// TwinCAT 3 PLC project tc_project_app
// ProgramVersion: 3.1.4026.24
// libraries:
//   Tc2_EtherCAT, * (Beckhoff Automation GmbH)
//   Tc2_MC2, * (Beckhoff Automation GmbH)
//   Tc2_Standard, * (Beckhoff Automation GmbH)
//   Tc2_SUPS, * (Beckhoff Automation GmbH)
//   Tc2_System, * (Beckhoff Automation GmbH)
//   Tc2_Utilities, * (Beckhoff Automation GmbH)
//   Tc3_EventLogger, * (Beckhoff Automation GmbH)
//   Tc3_MC2_AdvancedHoming, * (Beckhoff Automation GmbH)
//   Tc3_Module, * (Beckhoff Automation GmbH)
//   VisuDialogs, * (System)
// project tree:
//   DUTs/ E_AxisNames.TcDUT, E_PendantControl.TcDUT, E_SWLimitControl.TcDUT, ST_PendantControl.TcDUT
//   / GlobalTextList.TcGTLO, PlcTask.TcTTO, Visualization Manager.TcVMO (not stored)
//   GVLs/ GVL_APP.TcGVL, KeTop.TcGVL
//   POUs/Application_Specific/Applications/ Application_Template.TcPOU (not stored), Pendant.TcPOU
//   POUs/Application_Specific/Axes/ Axis1.TcPOU, Axis_Template.TcPOU, Pneumatics_Template.TcPOU (not stored)
//   POUs/Application_Specific/Groups/ GROUP_1.TcPOU, Group_Template.TcPOU
//   POUs/ MAIN.TcPOU, PANEL.TcPOU, SAFETY.TcPOU
//   tc_mca_std_lib/DUTs/Axis_Group_Structures/ ST_AxisGroupDescription.TcDUT, ST_AxisGroupFlag.TcDUT, ST_AxisGroupStruct.TcDUT
//   tc_mca_std_lib/DUTs/Axis_Structures/ ST_AxisConfig.TcDUT, ST_AxisControl.TcDUT, ST_AxisDescription.TcDUT, ST_AxisError.TcDUT, ST_AxisHomingConfig.TcDUT, ST_AxisInputs.TcDUT, ST_AxisPersistent.TcDUT, ST_AxisSPG.TcDUT, ST_AxisStatus.TcDUT, ST_AxisStruct.TcDUT
//   tc_mca_std_lib/DUTs/ E_AxisParameters.TcTLEO, E_AxisParameters.TcTLEO, E_HomingRoutines.TcDUT, E_RestorePosition.TcDUT, E_SafetyType.TcDUT, I_Axis.TcIO, E_SlitPairStatesV2.TcDUT, E_SlitPairStates.TcDUT, E_MotionFunctions.TcDUT, ST_McStatus.TcDUT
//   tc_mca_std_lib/DUTs/Panel_Infrastructure/ ST_ECB.TcDUT
//   tc_mca_std_lib/DUTs/Pneumatics/ E_PneumaticAxisErrors.TcDUT, E_PneumaticMode.TcDUT, ST_PneumaticAxisControl.TcDUT, ST_PneumaticAxisConfig.TcDUT, ST_PneumaticAxisInputs.TcDUT, ST_PneumaticAxisOutputs.TcDUT, ST_PneumaticAxisStatus.TcDUT, ST_PneumaticAxisStruct.TcDUT
//   tc_mca_std_lib/DUTs/Safety_Structures/ ST_DeviceDualChannelInput.TcDUT, ST_DeviceSingleChannelInput.TcDUT, ST_SafetyDescription.TcDUT, ST_SafetyGroup.TcDUT, ST_SafetyTargetDevice.TcDUT
//   tc_mca_std_lib/GVLs/ GVL.TcGVL, GVL_UnitStrings.TcGVL
//   tc_mca_std_lib/POUs/Motion/ FB_Axis.TcPOU, FB_AxisGroups.TcPOU, FB_SlitPair.TcPOU, FB_SlitPairV2.TcPOU, FB_SlitPairV3.TcPOU
//   tc_mca_std_lib/POUs/Motion/Homing/ FB_Homing.TcPOU
//   tc_mca_std_lib/POUs/Pneumatics/ FB_PneumaticAxis.TcPOU
//   tc_mca_std_lib/VISUs/ MainVisu.TcVIS, ParameterTextList.TcTLO, PneumaticsVisu.TcVIS
// real-time tasks:
//   TASK PlcTask: cycle T#10ms, priority 10, ADS port 351
// motion (NC):
//   TASK NC-Task 1 SAF: cycle T#2ms, priority 4, ADS port 501
//   TASK NC-Task 1 SVB: cycle T#10ms, priority 8, ADS port 511
//   AXIS Axis1 (id 1)
//     Dynamic: AccelerationMaximum=60, DecelerationMaximum=60, Acceleration=12, Deceleration=12, Jerk=42
//     Velo: RefSearch=5, RefSync=0.2, SlowManual=1, FastManual=5, Fast=9.091, Maximum=6.5
//     TargetPosControl: Range=0.25, Time=0.2
//     OtherSettings: AllowMotionCmdToSlave=true
//     encoder EncType=1
//       EncPara: ScaleFactorNumerator=20, ScaleFactorDenominator=12582912, Inverse=true
//         SoftEndMinControl: Range=-300
//         SoftEndMaxControl: Range=300
//     drive DrvType=5
//       DrvPara: Inverse=true
//         Analog: VeloReferenz=10.0001, TorqueSetpointScale=10, ScaleFactorActTorque=0.1
//         TimeComp: TaskDelayCycles=1
//     controller CtrType=1
//       CtrPara: PriorControlFactor=1
//         PosDiffControl: Range=2
//         Observer: BandWidth=20
// variable links:
//   tc_project_app Instance <-> NC-Task 1 SAF/Axes/Axis1
//     PlcTask Inputs/GVL.astAxes[1].Axis.NcToPlc <-> Outputs/ToPlc
//     PlcTask Outputs/GVL.astAxes[1].Axis.PlcToNc <-> Inputs/FromPlc

CONFIGURATION tc_project_app
    RESOURCE PLC ON TwinCAT3
        TASK PlcTask(INTERVAL := T#10ms, PRIORITY := 10);
        PROGRAM MAIN WITH PlcTask : MAIN;
        PROGRAM SAFETY WITH PlcTask : SAFETY;
        PROGRAM PANEL WITH PlcTask : PANEL;
    END_RESOURCE
END_CONFIGURATION

// ---- DUTs/E_AxisNames.TcDUT
{attribute 'qualified_only'}
{attribute 'to_string'}
TYPE E_AxisNames :
(
	None := 0,
	IncSlits_X_Translation := 1,
	IncSlits_Z_Translation :=2,
	IncSlits_North := 3,
	IncSlits_South := 4,
	IncSlits_East := 5,
	IncSlits_West := 6,
	Sample_Stack_X_Translation := 7,
	Sample_Stack_Y_Translation := 8,
	Tomography_Phi := 9,
	Tomography_Chi := 10,
	Tomography_Theta := 11,
	SampleEnv_ExtraAxes := 12,
	Camera_LensAdj := 13,
	Camera_FlipRot := 14, // check correct
	Camera_Tilt := 15, //check correct
	Sample_Stack_Z_Translation :=16,
	Sample_Stack_Z_Rotation :=17,
	Coll_North_X :=18,
	Coll_North_Y :=19,
	Coll_South_X :=20,
	Coll_South_Y :=21,
	PinholeSelector := 22,
	Monitor5 := 23,
	Slit_1_North := 24,
	Slit_1_South := 25,
	Slit_1_East := 26,
	Slit_1_West := 27,
	Slit_2_North := 28,
	Slit_2_South := 29,
	Slit_2_East := 30,
	Slit_2_West := 31,
	Slit_3_North := 32,
	Slit_3_South := 33,
	Slit_3_East := 34,
	Slit_3_West := 35,
	Slit_4_North := 36,
	Slit_4_South := 37,
	Slit_4_East := 38,
	Slit_4_West := 39,
	Slit_5_North := 40,
	Slit_5_South := 41,
	Slit_5_East := 42,
	Slit_5_West := 43
);
END_TYPE

// ---- DUTs/E_PendantControl.TcDUT
{attribute 'qualified_only'}
TYPE E_PendantControl :
(
	Default := 0,
	JogFwd := 33,
	JogBwd := 32,
	SmallTweakFwd := 19,
	SmallTweakBwd := 25,
	MediumTweakFwd := 45,
	MediumTweakBwd := 47,
	BigTweakFwd := 5,
	BigTweakBwd := 3,	
	AbsMove := 15,
	Stop := 12,
    SlowJogFwd := 38,
    SlowJogBwd := 36,
	WaitForAbsoluteFinish := 127,
	WaitForJogFinish := 128,
    WaitForTweakFinish := 129,
	Error := 150
);
END_TYPE

// ---- DUTs/E_SWLimitControl.TcDUT
{attribute 'qualified_only'}
TYPE E_SWLimitControl :
(
	Default := 0,
	WriteFwdLimit := 1,
	WriteBwdLimit := 2,
	EnableSWLimits := 3,
	DisableSWLimits := 4
);
END_TYPE

// ---- DUTs/ST_PendantControl.TcDUT
TYPE ST_PendantControl :
STRUCT
	fTargetPosition : LREAL;
	fVelocity : LREAL := 100;
	fFwdLimit : LREAL;
	fBwdLimit : LREAL;
	fLocalModeSpeedOverride : LREAL;
END_STRUCT
END_TYPE

// ---- tc_mca_std_lib/DUTs/Axis_Group_Structures/ST_AxisGroupDescription.TcDUT
TYPE ST_AxisGroupDescription :
STRUCT
	sGroupName : STRING(nMAX_AXIS_GROUP_NAME);
	iAxesInGroup : INT;
END_STRUCT
END_TYPE

// ---- tc_mca_std_lib/DUTs/Axis_Group_Structures/ST_AxisGroupFlag.TcDUT
TYPE ST_AxisGroupFlag :
STRUCT
	iError : INT;
	iDisabled : INT;
	iState : INT;
	bErrorFlag : BOOL;
	bDisabledFlag : BOOL;
	iNumberOfAxisInError : INT;
	iNumberOfAxisDisabled : INT;
END_STRUCT
END_TYPE

// ---- tc_mca_std_lib/DUTs/Axis_Group_Structures/ST_AxisGroupStruct.TcDUT
TYPE ST_AxisGroupStruct :
STRUCT
	aAxesInGroup : ARRAY[1..GVL.nMAX_AXES_PER_GROUP] OF INT :=[GVL.nMAX_AXES_PER_GROUP(0)];
	stDescription : ST_AxisGroupDescription;
	stFlag : ST_AxisGroupFlag;
END_STRUCT
END_TYPE

// ---- tc_mca_std_lib/DUTs/Axis_Structures/ST_AxisConfig.TcDUT
(*These are axis parameters that are set up during commissioning and
in theory don't neeed to be change as part of daily moving of axes.
For instance they may be changed due to poor parameter selection
or change of instrument configuration.*)
TYPE ST_AxisConfig :
STRUCT
    //Axis Parameters
    fOverride: LREAL := 100; //Controller override %, used a global scale for an axis in terms of velocity. Generally set to 100%.
    
    eRestorePosition: E_RestorePosition; //Restore position of incremental axis after loss of power to the CPU, 0=don't restore, 1=restore but don't home

    //Read and Write parameters
    eAxisParameters: E_AxisParameters; //Enumeration of axis parameters
	fWriteAxisBoolParameter: BOOL; //The Bool value to be writen to eAxisParameterNumber
    fWriteAxisParameter: LREAL; //The value to be writen to eAxisParameterNumber
    fReadAxisParameter: LREAL; //Read the current value of the selected eAxisParameterNumber

    

    // Read only MC parameters
    bReadMcParametersValid: BOOL:= FALSE;
    bReadMcParametersError: BOOL:= FALSE;
    fVelocityDefaultSlow: LREAL; //Read only - AxisVeloManSlow
    fVelocityDefaultFast: LREAL; //Read only - AxisVeloManFast
    
    fVeloMax: LREAL; //Read only - AxisMaxVelocity
    fMaxAcc: LREAL; //Read only - AxisMaximumAcceleration
    fMaxDec: LREAL; //Read only - AxisMaxDeceleration
    fDefaultAcc: LREAL; //Read only - AxisDefaultAcceleration
    fDefaultDec: LREAL; //Read only - AxisDefaultDeceleration
    bEnMinSoftPosLimit: BOOL; //Read only
    fMinSoftPosLimit: LREAL; //Read only
    bEnMaxSoftPosLimit: BOOL; //Read only
    fMaxSoftPosLimit: LREAL; //Read only
    bEnPositionLagMonitoring: BOOL; //Read only
    fMaxPosLagValue: LREAL; //Read only
    bEnTargetPositionMonitoring: BOOL; //Read only
    fTargetPositionWindow: LREAL; //Read only
END_STRUCT
END_TYPE

// ---- tc_mca_std_lib/DUTs/Axis_Structures/ST_AxisControl.TcDUT
(*These are parameters that are used to initiate axis movements
They are commands that are commonly used commands*)
TYPE ST_AxisControl :
STRUCT
    //Actions from controls system
    bExecute: BOOL; //Rising edge to execute some motion FB's
    bReset: BOOL; //Reset axis from Error state
    bStop: BOOL;
    bHalt: BOOL;
    bEnable: BOOL; //Enable axis drive
    bJogFwd: BOOL;
    bJogBwd: BOOL;
    bInterlockFwd: BOOL := FALSE; //Bit for interlocking motors in the positive direction
    bInterlockBwd: BOOL := FALSE; //Bit for interlocking motors in the negative direction
    eCommand: E_MotionFunctions;
    fVelocity: LREAL; //Velocity must be specified
    fJogVelocity: LREAL; //Jogging velocity
    fAcceleration: LREAL; //Not all FBs use, 0 is NC default
    fDeceleration: LREAL;
    fPosition: LREAL; //The position to move to for an absolute move and the amount to move in a relative move
	fRelativePosition: LREAL; //Position for relative moves
	fSetPosition : LREAL;
	bReinitialiseNcParameters : BOOL;
	bWaitBeforeEnable : BOOL:= FALSE; //Code to allow 'other things' to happen before enabling axis when working with autoenabledisable logic
	bReadyToEnable : BOOL; //trigger signal for the above
	
	bOverrideLimits : BOOL;
	
	bAutoEnableDisable : BOOL;
	
	bOverrideReadyToMove : BOOL;
	bExtReadyToMove : BOOL;
	tMoveFinishedDelay : TIME := T#1S;
END_STRUCT
END_TYPE

// ---- tc_mca_std_lib/DUTs/Axis_Structures/ST_AxisDescription.TcDUT
TYPE ST_AxisDescription :
STRUCT
	iGroupNumber : INT;
    sUnits : STRING := UNIT_mm;
END_STRUCT
END_TYPE

// ---- tc_mca_std_lib/DUTs/Axis_Structures/ST_AxisError.TcDUT

TYPE ST_AxisError:
STRUCT
//PLCopen function block errors
    nPowerErrorID: UDINT;
    nMoveAbsoluteErrorID: UDINT;
	nLocalMoveAbsoluteErrorID: UDINT;
    nMoveRelativeErrorID: UDINT;
	nLocalMoveRelativeErrorID: UDINT;
    nMoveVelocityErrorID: UDINT;
	nLocalMoveVelocityErrorID: UDINT;
    nMoveModuloErrorID: UDINT;
    nJogErrorID: UDINT;
    nHomeErrorID: UDINT;
    nHaltErrorID: UDINT;
    nResetErrorID: UDINT;
    nStopErrorID: UDINT;
    nGearInMultiMasterErrorID: UDINT;
    nGearOutErrorID: UDINT;
	nSetPositionErrorID : UDINT;
    fbWriteParameterErrorId: UDINT;
    fbReadParameterErrorId: UDINT;
//Error from the NC
    nNCErrorID : UDINT;
END_STRUCT
END_TYPE

// ---- tc_mca_std_lib/DUTs/Axis_Structures/ST_AxisHomingConfig.TcDUT
TYPE ST_AxisHomingConfig :
STRUCT
	fHomePosition: LREAL := 0; //The position that the axis should be set to once homing is completed
    fHomeFinishDistance: LREAL := 0; //Distrance that the axis should move back into the working zone after homing is finished
    eHomeSeq: E_HomingRoutines; //Homing sequence to perform
	fHomeAbsPosition : LREAL:= 0;
	fHomeMidRelativeMove : LREAL:= 1;
	
	bGoToFwdFirst : BOOL; //Takes priority over bwd bool, optional command to go to fwd limit before homing
	bGoToBwdFirst : BOOL; //optional command to go to bwd limit before homing
	bDoAbsoluteMoveAtEnd : BOOL;
	
	
	//General Advanced Homing Configuration
    bDisableDriveAccess: BOOL := TRUE; //Disables the drive access to drives. Standard for stepper motors. If supported in drive, can be set to FALSE, e.g. for AX5106.
    tTimeLimit: TIME; // Exceeding this time leads to the search procedure being aborted.
    fDistanceLimit: LREAL; // Exceeding this distance in relation to the start position leads to the search procedure being aborted.
    fTorqueLimit: LREAL; // The motor torque is limited to this value, in relation to the weight counterbalance that is possibly parameterized in the drive, in order to avoid mechanical damage.

    //Homing Configuration for Step Block
    fDetectionVelocityLimit: LREAL; // Velocity that must be fallen below for the DetectionVelocityTime in order to detect driving against the fixed stop.
    tDetectionVelocityTime: TIME; // Time for detecting the velocity undershoot when driving against the fixed stop.
    fLagLimit: LREAL; // Position lag value which, if exceeded, leads to detection of driving against the fixed stop.
	
	fHomingVelToCam: LREAL; //Read only - AxisCalibrationVelocityForward
    fHomingVelFromCam: LREAL; //Read only - AxisCalibrationVelocityBackward
END_STRUCT
END_TYPE

// ---- tc_mca_std_lib/DUTs/Axis_Structures/ST_AxisInputs.TcDUT
TYPE ST_AxisInputs :
STRUCT
    bLimitFwd AT %I*: BOOL;
    bLimitBwd AT %I*: BOOL;
    bHomeSensor AT %I*: BOOL; //Reference signal for homing
	bPermit : BOOL :=TRUE; //Permit signal to block moves if safety does not allow - used to prevent queuing commands, default as true, set in axis prog
	bAllowRemoteControl : BOOL;
END_STRUCT
END_TYPE

// ---- tc_mca_std_lib/DUTs/Axis_Structures/ST_AxisPersistent.TcDUT
TYPE ST_AxisPersistent :
STRUCT RETAIN
    //Settings for restoring positions on power off
    fPositionAtShutdown: LREAL; //The position that the axis was at when CPU shut down
    fEncoderBiasAtShutdown: LREAL; //Encoder position BIAS value when CPU shut down
    bMovingAtShutdown: BOOL; //True if the axis was moving at shutdown, False otherwise
END_STRUCT
END_TYPE

// ---- tc_mca_std_lib/DUTs/Axis_Structures/ST_AxisSPG.TcDUT
TYPE ST_AxisSPG :
STRUCT
	EnableSPG : BOOL;
	DisableSPG : BOOL;
	
	
	Position : LREAL;
	Velocity : LREAL;
	VelocityStandstillThreshold : LREAL := 0; //Can be zero
	Acceleration : LREAL;
	Direction : DINT;
	OverrideDirection : BOOL := FALSE; //TRUE for manual direction feed otherwise calculated in FB_AXIS
END_STRUCT
END_TYPE

// ---- tc_mca_std_lib/DUTs/Axis_Structures/ST_AxisStatus.TcDUT
TYPE ST_AxisStatus :
STRUCT
    //Outputs & Status
    bAxisInitialized: BOOL := FALSE; //True when all parameters from actReadMcParameters are valid
    bEnabled: BOOL; //Axis drive enabled
    bCommandAborted: BOOL; //Command aborted output of the eCommand function blocks
    bBusy: BOOL; //Axis busy (eCommand function block is active)
    bDone: BOOL; //Last eCommand function block executed successfully;
    //bDone will also be set with the InGear and InVelocity outputs
    //When InVelocity is set, fbMoveVelocity is still acitve, which is reflected by the bBusy status
    bInVelocity: BOOL; //MC_MoveVelocity has reached target velocity; will stay true until the movement stops
    bHomed: BOOL; //Axis homed
    bMoving: BOOL; //Moving state from the NC
    bMovingForward: BOOL; //Moving forward indicator from NC
    bMovingBackward: BOOL; //Moving backward indicator from NC
    bInTargetPosition: BOOL; //In target position bit from AxisStatus()
    bFwEnabled: BOOL; //Positive movement of axis is enabled/disabled
    bBwEnabled: BOOL; //Negative movement of axis is enabled/disabled
    bInterlockedFwd: BOOL; //Axis interlocked in the postive direction
    bInterlockedBwd: BOOL; //Axis interlocked in the negative direction
	bSTOActive AT %I*: BOOL;
	bInHomingSeq : BOOL; //Prehoming limit move in progress

    fActPosition: LREAL; //Actual position value


    fActVelocity: LREAL; //Actual velocity
    bError: BOOL; //Reserved for NC error states that actually block motion
	bMcError : BOOL; //Reserved for errors generated for MC PLC function blocks
    nErrorID: UDINT; //NC errorID
	nMcErrorID: UDINT;//Last motion function block errorID
	
	bReadyToMove : BOOL;
	bMoveRequested : BOOL;
	bMoveInProgress : BOOL;
	
	SPGEnabled : BOOL;
	
	bPositionRestored : BOOL;
	
	
	messageString : STRING; //FB_Axis Execution messages
	appMessageString : STRING; //Message string reserved for application specific functionality
	errorString : STRING; //NC Converted values as a lookup table (but translated
END_STRUCT
END_TYPE

// ---- tc_mca_std_lib/DUTs/Axis_Structures/ST_AxisStruct.TcDUT
TYPE ST_AxisStruct :
STRUCT
    stControl: ST_AxisControl;
    stStatus: ST_AxisStatus;
    stConfig: ST_AxisConfig;
    stError: ST_AxisError;
    stInputs: ST_AxisInputs;
    stDescription: ST_AxisDescription;
	stHomingConfig : ST_AxisHomingConfig;
	stSpg : ST_AxisSPG;
    //The NC axis link to the hardware that is controlling
    Axis: AXIS_REF;
	Commissioning : BOOL :=FALSE;
END_STRUCT
END_TYPE

// ---- tc_mca_std_lib/DUTs/E_AxisParameters.TcTLEO
{attribute 'qualified_only'}
{attribute 'strict'}
TYPE E_AxisParameters :
(
//PLCopen specific parameters Index-Group 0x4000 + ID
    CommandedPosition := 1, //lreal taken from NcToPlc
    SWLimitForward := 2, //lreal IndexOffset= 16#0001_000E
    SWLimitBackward := 3, //lreal IndexOffset= 16#0001_000D
    EnableLimitForward := 4, //bool IndexOffset= 16#0001_000C
    EnableLimitBackward := 5, //bool IndexOffset= 16#0001_000B
    EnablePositionLagMonitoring := 6, //bool IndexOffset= 16#0002_0010
    MaxPositionLag := 7, //lreal IndexOffset= 16#0002_0012
    AxisMaxVelocity := 8, //lreal IndexOffset= 16#0000_0027
    ActualVelocity := 10, //lreal taken from NcToPlc
    CommandedVelocity := 11, //lreal taken from NcToPlc
    AxisDefaultAcceleration := 12, //lreal IndexOffset= 16#0000_0101
    AxisDefaultDeceleration := 14, //lreal IndexOffset= 16#0000_0102
    AxisDefaultJerk := 16, //lreal IndexOffset= 16#0000_0103

//Beckhoff specific parameters Index-Group 0x4000 + ID
    AxisId := 1000, //lreal IndexOffset= 16#0000_0001
    AxisManualVelocitySlow := 1001, //lreal IndexOffset= 16#0000_0008
    AxisManualVelocityFast := 1002, //lreal IndexOffset= 16#0000_0009
    AxisRapidTraverseVelocity := 1009, //lreal IndexOffset= 16#0000_000A
    AxisVelocityToCam := 1012, //lreal IndexOffset= 16#0000_0006
    AxisVelocityFromCam := 1013, //lreal IndexOffset= 16#0000_0007
    AxisJogIncrementForward := 1014, //lreal IndexOffset= 16#0000_0018
    AxisJogIncrementBackward := 1015, //lreal IndexOffset= 16#0000_0019
    MaxPositionLagFilterTime := 1022, //lreal IndexOffset= 16#0002_0013
    AxisEnPositionRangeMonitoring := 1023, //bool IndexOffset= 16#0000_000F
    AxisPositionRangeWindow := 1024, //lreal IndexOffset= 16#0000_0010
    AxisEnTargetPositionMonitoring:= 1025, //bool IndexOffset= 16#0000_0015
    AxisTargetPositionWindow := 1026, //lreal IndexOffset= 16#0000_0016
    AxisTargetPositionMonitoringTime := 1027, //lreal IndexOffset= 16#0000_0017
    AxisEnInTargetTimeout := 1028, //bool IndexOffset= 16#0000_0029
    AxisInTargetTimeout := 1029, //lreal IndexOffset= 16#0000_002A
    AxisEnMotionMonitoring := 1030, //bool IndexOffset= 16#0000_0011
    AxisMotionMonitoringWindow := 1031, //lreal IndexOffset= 16#0000_0028
    AxisMotionMonitoringTime := 1032, //lreal IndexOffset= 16#0000_0012
    AxisDelayTimeVeloPosition := 1033, //lreal IndexOffset= 16#0000_0104
    AxisEnLoopingDistance := 1034, //bool IndexOffset= 16#0000_0013
    AxisLoopingDistance := 1035, //lreal IndexOffset= 16#0000_0014
    AxisEnBacklashCompensation := 1036, //bool IndexOffset= 16#0000_002B
    AxisBacklash := 1037, //lreal IndexOffset= 16#0000_002C
    AxisEnDataPersistence := 1038, //bool IndexOffset= 16#0000_0030
    AxisRefVeloOnRefOutput := 1039, //lreal IndexOffset= 16#0003_0101
    AxisOverrideType := 1040, //lreal IndexOffset= 16#0000_0105
    //new since 4/2007
    AxisEncoderOffset := 1042, //lreal IndexOffset= 16#0001_0007
    AxisEncoderDirectionInverse := 1043, //bool IndexOffset= 16#0001_0008
    AxisEncoderMask := 1044, //dword IndexOffset= 16#0001_0015
    AxisEncoderModuloValue := 1045, //lreal IndexOffset= 16#0001_0009
    AxisModuloToleranceWindow := 1046, //lreal IndexOffset= 16#0001_001B
    AxisEnablePosCorrection := 1047, //bool IndexOffset= 16#0001_0016
    AxisPosCorrectionFilterTime := 1048, //lreal IndexOffset= 16#0001_0017
    //new since 1/2010
    AxisUnitInterpretation := 1049, //lreal IndexOffset= 16#0000_0026
    AxisMotorDirectionInverse := 1050, //bool  IndexOffset= 16#0003_0006
    //new since 1/2011
    AxisCycleTime := 1051, //lreal IndexOffset= 16#0000_0004
    //new since 5/2011
    AxisFastStopSignalType := 1052, //dword IndexOffset= 16#0000_001E
    AxisFastAcc := 1053, //lreal IndexOffset= 16#0000_010A
    AxisFastDec := 1054, //lreal IndexOffset= 16#0000_010B
    AxisFastJerk := 1055, //lreal IndexOffset= 16#0000_010C
    // new since 1/2012 *)
    AxisEncoderScalingNumerator := 1056, //lreal IndexOffset= 16#0001_0023 - available in Tc3
    AxisEncoderScalingDenominator := 1057, //lreal IndexOffset= 16#0001_0024 - available in Tc3
    (* new since 7/2016 *)
    AxisMaximumAcceleration := 1058, //lreal IndexOffset= 16#0000_00F1
    AxisMaximumDeceleration := 1059, //lreal IndexOffset= 16#0000_00F2
    AxisVeloJumpFactor := 1060, //lreal IndexOffset= 16#0000_0106
    AxisToleranceBallAuxAxis := 1061, //lreal IndexOffset= 16#0000_0108
    AxisMaxPositionDeviationAuxAxis := 1062, //lreal IndexOffset= 16#0000_0109
    AxisErrorPropagationMode := 1063, //dword IndexOffset= 16#0000_001A
    AxisErrorPropagationDelay := 1064, //lreal IndexOffset= 16#0000_001B
    AxisCoupleSlaveToActualValues := 1065, //bool IndexOffset= 16#0000_001C
    AxisAllowMotionCmdToSlaveAxis := 1066, //bool IndexOffset= 16#0000_0020
    AxisAllowMotionCmdToExtSetAxis := 1067, //bool IndexOffset= 16#0000_0021
    AxisEncoderSubMask := 1068, //dword IndexOffset= 16#0001_0108
    AxisEncoderReferenceSystem := 1069, //dword IndexOffset= 16#0001_0019
    AxisEncoderPositionFilterPT1 := 1070, //lreal IndexOffset= 16#0001_0010
    AxisEncoderVelocityFilterPT1 := 1071, //lreal IndexOffset= 16#0001_0011
    AxisEncoderAccelerationFilterPT1 := 1072, //lreal IndexOffset= 16#0001_0012
    AxisEncoderMode := 1073, //dword IndexOffset= 16#0001_000A
    AxisEncoderHomingInvDirCamSearch := 1074, //bool IndexOffset= 16#0001_0101
    AxisEncoderHomingInvDirSyncSearch := 1075, //bool IndexOffset= 16#0001_0102
    AxisEncoderHomingCalibValue := 1076, //lreal IndexOffset= 16#0001_0103
    AxisEncoderReferenceMode := 1077, //dword IndexOffset= 16#0001_0107
    AxisRefVeloOutputRatio := 1078, //lreal IndexOffset= 16#0003_0102
    AxisDrivePositionOutputScaling := 1079, //lreal IndexOffset= 16#0003_0109
    AxisDriveVelocityOutputScaling := 1080, //lreal IndexOffset= 16#0003_0105
    AxisDriveVelocityOutputDelay := 1081, //lreal IndexOffset= 16#0003_010D
    AxisDriveMinOutputLimitation := 1082, //lreal IndexOffset= 16#0003_000B
    AxisDriveMaxOutputLimitation := 1083, //lreal IndexOffset= 16#0003_000C
    AxisTorqueInputScaling := 1084, //lreal IndexOffset= 16#0003_0031 - available in Tc3
    AxisTorqueInputFilterPT1 := 1085, //lreal IndexOffset= 16#0003_0032 - available in Tc3
    AxisTorqueDerivationInputFilterPT1 := 1086, //lreal IndexOffset= 16#0003_0033 - available in Tc3
    AxisTorqueOutputScaling := 1087, //lreal IndexOffset= 16#0003_010B
    AxisTorqueOutputDelay := 1088, //lreal IndexOffset= 16#0003_010F
    AxisAccelerationOutputScaling := 1089, //lreal IndexOffset= 16#0003_010A
    AxisAccelerationOutputDelay := 1090, //lreal IndexOffset= 16#0003_010E
    AxisDrivePositionOutputSmoothFilterType := 1091, //dword IndexOffset= 16#0003_0110
    AxisDrivePositionOutputSmoothFilterTime := 1092, //lreal IndexOffset= 16#0003_0111
    AxisDrivePositionOutputSmoothFilterOrder := 1093, //dword IndexOffset= 16#0003_0112
    AxisDriveMode := 1094, //dword IndexOffset= 16#0003_000A
    AxisDriftCompensationOffset := 1095, //lreal IndexOffset= 16#0003_0104
    AxisPositionControlKv := 1096, //lreal IndexOffset= 16#0002_0102
    AxisCtrlVelocityPreCtrlWeight := 1097, //lreal IndexOffset= 16#0002_000B
    AxisControllerMode := 1098, //dword IndexOffset= 16#0002_000A
    AxisCtrlAutoOffset := 1099, //bool IndexOffset= 16#0002_0110
    AxisCtrlAutoOffsetTimer := 1100, //lreal IndexOffset= 16#0002_0115
    AxisCtrlAutoOffsetLimit := 1101, //lreal IndexOffset= 16#0002_0114
    AxisSlaveCouplingControlKcp := 1102, //lreal IndexOffset= 16#0002_010F
    AxisCtrlOutputLimit := 1103, //lreal IndexOffset= 16#0002_0100

//Beckhoff specific axis status information - READ ONLY Index-Group 0x4100 + ID
    AxisTargetPosition := 2000, //lreal IndexOffset= 16#0000_0013
    AxisRemainingTimeToGo := 2001, //lreal IndexOffset= 16#0000_0014
    AxisRemainingDistanceToGo := 2002, //lreal IndexOffset= 16#0000_0022, 16#0000_0042

//Beckhoff specific axis functions
    //read/write gear ratio of a slave
    AxisGearRatio := 3000, //lreal read: IndexGroup=0x4100+ID, IdxOffset=16#0000_0022,
                                 //write:IndexGroup=0x4200+ID, IdxOffset=16#0000_0042

//Beckhoff specific other parameters
    //new since 1/2011
    NcSafCycleTime := 4000, //lreal IndexOffset= 16#0000_0010
    NcSvbCycleTime := 4001 //lreal IndexOffset= 16#0000_0012

);
END_TYPE

// ---- tc_mca_std_lib/DUTs/E_AxisParameters.TcTLEO
{attribute 'qualified_only'}
{attribute 'strict'}
TYPE E_AxisParameters :
(
//PLCopen specific parameters Index-Group 0x4000 + ID
    CommandedPosition := 1, //lreal taken from NcToPlc
    SWLimitForward := 2, //lreal IndexOffset= 16#0001_000E
    SWLimitBackward := 3, //lreal IndexOffset= 16#0001_000D
    EnableLimitForward := 4, //bool IndexOffset= 16#0001_000C
    EnableLimitBackward := 5, //bool IndexOffset= 16#0001_000B
    EnablePositionLagMonitoring := 6, //bool IndexOffset= 16#0002_0010
    MaxPositionLag := 7, //lreal IndexOffset= 16#0002_0012
    AxisMaxVelocity := 8, //lreal IndexOffset= 16#0000_0027
    ActualVelocity := 10, //lreal taken from NcToPlc
    CommandedVelocity := 11, //lreal taken from NcToPlc
    AxisDefaultAcceleration := 12, //lreal IndexOffset= 16#0000_0101
    AxisDefaultDeceleration := 14, //lreal IndexOffset= 16#0000_0102
    AxisDefaultJerk := 16, //lreal IndexOffset= 16#0000_0103

//Beckhoff specific parameters Index-Group 0x4000 + ID
    AxisId := 1000, //lreal IndexOffset= 16#0000_0001
    AxisManualVelocitySlow := 1001, //lreal IndexOffset= 16#0000_0008
    AxisManualVelocityFast := 1002, //lreal IndexOffset= 16#0000_0009
    AxisRapidTraverseVelocity := 1009, //lreal IndexOffset= 16#0000_000A
    AxisVelocityToCam := 1012, //lreal IndexOffset= 16#0000_0006
    AxisVelocityFromCam := 1013, //lreal IndexOffset= 16#0000_0007
    AxisJogIncrementForward := 1014, //lreal IndexOffset= 16#0000_0018
    AxisJogIncrementBackward := 1015, //lreal IndexOffset= 16#0000_0019
    MaxPositionLagFilterTime := 1022, //lreal IndexOffset= 16#0002_0013
    AxisEnPositionRangeMonitoring := 1023, //bool IndexOffset= 16#0000_000F
    AxisPositionRangeWindow := 1024, //lreal IndexOffset= 16#0000_0010
    AxisEnTargetPositionMonitoring:= 1025, //bool IndexOffset= 16#0000_0015
    AxisTargetPositionWindow := 1026, //lreal IndexOffset= 16#0000_0016
    AxisTargetPositionMonitoringTime := 1027, //lreal IndexOffset= 16#0000_0017
    AxisEnInTargetTimeout := 1028, //bool IndexOffset= 16#0000_0029
    AxisInTargetTimeout := 1029, //lreal IndexOffset= 16#0000_002A
    AxisEnMotionMonitoring := 1030, //bool IndexOffset= 16#0000_0011
    AxisMotionMonitoringWindow := 1031, //lreal IndexOffset= 16#0000_0028
    AxisMotionMonitoringTime := 1032, //lreal IndexOffset= 16#0000_0012
    AxisDelayTimeVeloPosition := 1033, //lreal IndexOffset= 16#0000_0104
    AxisEnLoopingDistance := 1034, //bool IndexOffset= 16#0000_0013
    AxisLoopingDistance := 1035, //lreal IndexOffset= 16#0000_0014
    AxisEnBacklashCompensation := 1036, //bool IndexOffset= 16#0000_002B
    AxisBacklash := 1037, //lreal IndexOffset= 16#0000_002C
    AxisEnDataPersistence := 1038, //bool IndexOffset= 16#0000_0030
    AxisRefVeloOnRefOutput := 1039, //lreal IndexOffset= 16#0003_0101
    AxisOverrideType := 1040, //lreal IndexOffset= 16#0000_0105
    //new since 4/2007
    AxisEncoderOffset := 1042, //lreal IndexOffset= 16#0001_0007
    AxisEncoderDirectionInverse := 1043, //bool IndexOffset= 16#0001_0008
    AxisEncoderMask := 1044, //dword IndexOffset= 16#0001_0015
    AxisEncoderModuloValue := 1045, //lreal IndexOffset= 16#0001_0009
    AxisModuloToleranceWindow := 1046, //lreal IndexOffset= 16#0001_001B
    AxisEnablePosCorrection := 1047, //bool IndexOffset= 16#0001_0016
    AxisPosCorrectionFilterTime := 1048, //lreal IndexOffset= 16#0001_0017
    //new since 1/2010
    AxisUnitInterpretation := 1049, //lreal IndexOffset= 16#0000_0026
    AxisMotorDirectionInverse := 1050, //bool  IndexOffset= 16#0003_0006
    //new since 1/2011
    AxisCycleTime := 1051, //lreal IndexOffset= 16#0000_0004
    //new since 5/2011
    AxisFastStopSignalType := 1052, //dword IndexOffset= 16#0000_001E
    AxisFastAcc := 1053, //lreal IndexOffset= 16#0000_010A
    AxisFastDec := 1054, //lreal IndexOffset= 16#0000_010B
    AxisFastJerk := 1055, //lreal IndexOffset= 16#0000_010C
    // new since 1/2012 *)
    AxisEncoderScalingNumerator := 1056, //lreal IndexOffset= 16#0001_0023 - available in Tc3
    AxisEncoderScalingDenominator := 1057, //lreal IndexOffset= 16#0001_0024 - available in Tc3
    (* new since 7/2016 *)
    AxisMaximumAcceleration := 1058, //lreal IndexOffset= 16#0000_00F1
    AxisMaximumDeceleration := 1059, //lreal IndexOffset= 16#0000_00F2
    AxisVeloJumpFactor := 1060, //lreal IndexOffset= 16#0000_0106
    AxisToleranceBallAuxAxis := 1061, //lreal IndexOffset= 16#0000_0108
    AxisMaxPositionDeviationAuxAxis := 1062, //lreal IndexOffset= 16#0000_0109
    AxisErrorPropagationMode := 1063, //dword IndexOffset= 16#0000_001A
    AxisErrorPropagationDelay := 1064, //lreal IndexOffset= 16#0000_001B
    AxisCoupleSlaveToActualValues := 1065, //bool IndexOffset= 16#0000_001C
    AxisAllowMotionCmdToSlaveAxis := 1066, //bool IndexOffset= 16#0000_0020
    AxisAllowMotionCmdToExtSetAxis := 1067, //bool IndexOffset= 16#0000_0021
    AxisEncoderSubMask := 1068, //dword IndexOffset= 16#0001_0108
    AxisEncoderReferenceSystem := 1069, //dword IndexOffset= 16#0001_0019
    AxisEncoderPositionFilterPT1 := 1070, //lreal IndexOffset= 16#0001_0010
    AxisEncoderVelocityFilterPT1 := 1071, //lreal IndexOffset= 16#0001_0011
    AxisEncoderAccelerationFilterPT1 := 1072, //lreal IndexOffset= 16#0001_0012
    AxisEncoderMode := 1073, //dword IndexOffset= 16#0001_000A
    AxisEncoderHomingInvDirCamSearch := 1074, //bool IndexOffset= 16#0001_0101
    AxisEncoderHomingInvDirSyncSearch := 1075, //bool IndexOffset= 16#0001_0102
    AxisEncoderHomingCalibValue := 1076, //lreal IndexOffset= 16#0001_0103
    AxisEncoderReferenceMode := 1077, //dword IndexOffset= 16#0001_0107
    AxisRefVeloOutputRatio := 1078, //lreal IndexOffset= 16#0003_0102
    AxisDrivePositionOutputScaling := 1079, //lreal IndexOffset= 16#0003_0109
    AxisDriveVelocityOutputScaling := 1080, //lreal IndexOffset= 16#0003_0105
    AxisDriveVelocityOutputDelay := 1081, //lreal IndexOffset= 16#0003_010D
    AxisDriveMinOutputLimitation := 1082, //lreal IndexOffset= 16#0003_000B
    AxisDriveMaxOutputLimitation := 1083, //lreal IndexOffset= 16#0003_000C
    AxisTorqueInputScaling := 1084, //lreal IndexOffset= 16#0003_0031 - available in Tc3
    AxisTorqueInputFilterPT1 := 1085, //lreal IndexOffset= 16#0003_0032 - available in Tc3
    AxisTorqueDerivationInputFilterPT1 := 1086, //lreal IndexOffset= 16#0003_0033 - available in Tc3
    AxisTorqueOutputScaling := 1087, //lreal IndexOffset= 16#0003_010B
    AxisTorqueOutputDelay := 1088, //lreal IndexOffset= 16#0003_010F
    AxisAccelerationOutputScaling := 1089, //lreal IndexOffset= 16#0003_010A
    AxisAccelerationOutputDelay := 1090, //lreal IndexOffset= 16#0003_010E
    AxisDrivePositionOutputSmoothFilterType := 1091, //dword IndexOffset= 16#0003_0110
    AxisDrivePositionOutputSmoothFilterTime := 1092, //lreal IndexOffset= 16#0003_0111
    AxisDrivePositionOutputSmoothFilterOrder := 1093, //dword IndexOffset= 16#0003_0112
    AxisDriveMode := 1094, //dword IndexOffset= 16#0003_000A
    AxisDriftCompensationOffset := 1095, //lreal IndexOffset= 16#0003_0104
    AxisPositionControlKv := 1096, //lreal IndexOffset= 16#0002_0102
    AxisCtrlVelocityPreCtrlWeight := 1097, //lreal IndexOffset= 16#0002_000B
    AxisControllerMode := 1098, //dword IndexOffset= 16#0002_000A
    AxisCtrlAutoOffset := 1099, //bool IndexOffset= 16#0002_0110
    AxisCtrlAutoOffsetTimer := 1100, //lreal IndexOffset= 16#0002_0115
    AxisCtrlAutoOffsetLimit := 1101, //lreal IndexOffset= 16#0002_0114
    AxisSlaveCouplingControlKcp := 1102, //lreal IndexOffset= 16#0002_010F
    AxisCtrlOutputLimit := 1103, //lreal IndexOffset= 16#0002_0100

//Beckhoff specific axis status information - READ ONLY Index-Group 0x4100 + ID
    AxisTargetPosition := 2000, //lreal IndexOffset= 16#0000_0013
    AxisRemainingTimeToGo := 2001, //lreal IndexOffset= 16#0000_0014
    AxisRemainingDistanceToGo := 2002, //lreal IndexOffset= 16#0000_0022, 16#0000_0042

//Beckhoff specific axis functions
    //read/write gear ratio of a slave
    AxisGearRatio := 3000, //lreal read: IndexGroup=0x4100+ID, IdxOffset=16#0000_0022,
                                 //write:IndexGroup=0x4200+ID, IdxOffset=16#0000_0042

//Beckhoff specific other parameters
    //new since 1/2011
    NcSafCycleTime := 4000, //lreal IndexOffset= 16#0000_0010
    NcSvbCycleTime := 4001 //lreal IndexOffset= 16#0000_0012

);
END_TYPE

// ---- tc_mca_std_lib/DUTs/E_HomingRoutines.TcDUT
{attribute 'qualified_only'}
{attribute 'strict'}
TYPE E_HomingRoutines :
(
    eNoHoming := 0,

    //0X: LIMIT Switch
    //Home to bBwdLimit, record position on first approach
    eHomeToLimit_Bwd := 1,
    //Home to bFwdLimit, record position on first approach
    eHomeToLimit_Fwd := 2,
    //Find bBwdLimit (using towardsCam speed), then reverse direction looking FOR falling edge (using fromCam speed)
    //eHomeToLimit_Bwd_2Speeds := 3,
    //Find bFwdLimit (using towardsCam speed), then reverse direction looking for falling edge (using fromCam speed)
    //eHomeToLimit_Fwd_2Speeds := 4,

    //1X: Home Sensor
    //Home to bHome in Bwd direction (will reverse direction if limit hit), record position on first approach
    eHomeToRef_Bwd := 11,
    //Home to bHome in Fwd direction (will reverse direction if limit hit), record position on first approach
    eHomeToRef_Fwd := 12,
    //Find bHome in Bwd direction (using towardsCam speed) then reverse direction looking for falling edge (using fromCam speed), will reverse direction if limit hit
    eHomeToRef_Bwd_Fast := 13,
    //Find bHome in Fwd direction (using towardsCam speed) then reverse direction looking for falling edge (using fromCam speed), will reverse direction if limit hit
    eHomeToRef_Fwd_Fast := 14,

    //2X: Enc Pulse
    //Home to EncRefPulse in Bwd direction (used for single turn rotary axis without limit switches)
    eHomeToEncPulse_Bwd := 21,
    //Home to EncRefPulse in Fwd direction (used for single turn rotary axis without limit switches)
    eHomeToEncPulse_Fwd := 22,
    //Home to EncRefPulse via bBwdLimit (using towardsCam speed), then reverse direction looking for falling edge on ref pulse (using fromCam speed)
    eHomeToEncPulse_viaBwdLimit := 23,
    //Home to EncRefPulse via bFwdLimit (using towardsCam speed), then reverse direction looking for falling edge on ref pulse (using fromCam speed)
    eHomeToEncPulse_viaFwdLimit := 24,
	
	//Fast search for EncRefPulse in BWD direction (using towards cam) then moves off and refinds slower (From cam)
	eHomeToEncPulse_BWD_FAST := 25,
	//Fast search for EncRefPulse in FWD direction (using towards cam) then moves off and refinds slower (From cam)
	eHomeToEncPulse_FWD_FAST := 26,

    //3X: Home To Mechanical Block (Lag based StepBlockDetection)
    //Home towards a mechanical block in Bwd direction
    eHomeToBlock_Bwd := 30,
    //Home towards a mechanical block in Fwd direction
    eHomeToBlock_Fwd := 31,

    //9X: Software
    eHomeDirect := 90 //Set position directly to fHomePosition
) := eHomeDirect;
END_TYPE

// ---- tc_mca_std_lib/DUTs/E_RestorePosition.TcDUT
{attribute 'qualified_only'}
{attribute 'strict'}
TYPE E_RestorePosition :
(
    eDontRestore :=0,
    eRestoreWithoutHome := 1 //Redefined the position of the axis to that when the power was lost
);
END_TYPE

// ---- tc_mca_std_lib/DUTs/E_SafetyType.TcDUT
{attribute 'qualified_only'}
{attribute 'strict'}
TYPE E_SafetyType :
(
	eSingleChannel := 0
);
END_TYPE

// ---- tc_mca_std_lib/DUTs/E_SlitPairStatesV2.TcDUT

{attribute 'qualified_only'}
{attribute 'strict'}
TYPE E_SlitPairStatesV2 :
(
    eInit := 0,
    eEnableRealGenerators,
    eDisableRealGenerators,
    eEnableVirtualGenerators,
    eDisableVirtualGenerators,
    eWaitForVirtualMoveDone,
    eWaitForRealMoveDone,
    eError,
    eOperational,
    eWaitForVirtualHomed,
    eWaitForRealHomed,
    eCheckRealAxisGeneratorsEnabled,
    eCheckVirtualAxisGeneratorsEnabled
);
END_TYPE

// ---- tc_mca_std_lib/DUTs/Panel_Infrastructure/ST_ECB.TcDUT
TYPE ST_ECB :
STRUCT
	Status AT %I* : BOOL;
	Reset AT %Q* : BOOL;
	Name : STRING;
	Description : STRING;
END_STRUCT
END_TYPE

// ---- tc_mca_std_lib/DUTs/Pneumatics/E_PneumaticAxisErrors.TcDUT
{attribute 'qualified_only'}
{attribute 'strict'}
TYPE E_PneumaticAxisErrors :
(
    eNoError := 0,
    eExtractTimedOut := 1, //Extraction movement not done in expected time
    eRetractTimedOut := 2, //Retraction movement not done in expected time
    eNotMovingExtract := 3, //Extract command not executed, cylinder stays in place
    eNotMovingRetract := 4, //Retract command not executed, cylinder stays in place
    eInterlockOn := 5, //Interlock signal on, cylinder retracts to Limit Bwd
    eNoPSSPermit := 6, //Permit signal lost, cylinder retracts to Limit Bwd
    eAirPressureError := 7 //Air pressure signal out of range
):= eNoError;
END_TYPE

// ---- tc_mca_std_lib/DUTs/Pneumatics/E_PneumaticMode.TcDUT
{attribute 'qualified_only'}
{attribute 'strict'}
TYPE E_PneumaticMode :
(   eSingleSolenoidControl := 0, //Single solenoid valve with spring return
    eReset := 1,
    eError := 2
):= eSingleSolenoidControl;
END_TYPE

// ---- tc_mca_std_lib/DUTs/Pneumatics/ST_PneumaticAxisControl.TcDUT
TYPE ST_PneumaticAxisControl :
STRUCT
    bExtend: BOOL; //Variable to control solenoid valve from PLC
    bRetract: BOOL; //Variable to control solenoid valve from PLC
    bInterlock: BOOL; //Input interlock signal for the movement
    bReset: BOOL; //Reset signal from EPICS
END_STRUCT
END_TYPE

// ---- tc_mca_std_lib/DUTs/Pneumatics/ST_PneumaticAxisConfig.TcDUT
TYPE ST_PneumaticAxisConfig :
STRUCT
    nTimeToExtend: INT; //User defined time for the cylider to extract in seconds
    nTimeToRetract: INT; //User defined time for the cylinder to retract in seconds
END_STRUCT
END_TYPE

// ---- tc_mca_std_lib/DUTs/Pneumatics/ST_PneumaticAxisInputs.TcDUT
TYPE ST_PneumaticAxisInputs :
STRUCT
    bEndSwitchFwd AT %I*: BOOL; //End Switch Fwd input
    bEndSwitchBwd AT %I*: BOOL; //End Switch Bwd input
    bSolenoidActive AT %I*: BOOL; //Solenoid valve Extend Input (for single solenoid)
    bPSSPermit AT %I*: BOOL; //Input signal from PSS for the movement
    bPressureExtend AT %I*: BOOL; //Input signal of air pressure for cyclinder extraction
    bPressureRetract AT %I*: BOOL; //Input signal of air pressure for cylinder retraction
    nAirPressureValve AT %I*: REAL; //Input signal of air pressure for pneumatic valve
    bOpenManual AT %I*: BOOL; //Push button input to extend cylinder
    bCloseManual AT %I*: BOOL; //Push button input to retract the cylinder
END_STRUCT
END_TYPE

// ---- tc_mca_std_lib/DUTs/Pneumatics/ST_PneumaticAxisOutputs.TcDUT
TYPE ST_PneumaticAxisOutputs :
STRUCT
    bEndSwitchFwdOn AT %Q*: BOOL; //End Switch Fwd power output
    bEndSwitchBwdOn AT %Q*: BOOL; //End Switch Bwd power output
    bValveOn AT %Q*: BOOL; //Output of the solenoid valve (for single solenoid)
    bPressureExtendOn AT %Q*: BOOL; //Power output for air pressure switch
    bPressureRetractOn AT %Q*: BOOL; //Power output for air pressure switch
    fAirPressureOn AT %Q*: REAL; //Power output for analog pressure sensor
END_STRUCT
END_TYPE

// ---- tc_mca_std_lib/DUTs/Pneumatics/ST_PneumaticAxisStatus.TcDUT
TYPE ST_PneumaticAxisStatus :
STRUCT
    bExtending: BOOL; //Extending movement status
    bRetracting: BOOL; //Retraction movement status
    bExtended: BOOL; //Cylinder extracted status
    bRetracted: BOOL; //Cylinder retracted status
    nTimeElapsedExtend: INT; //Elapsed time while extracting cylinder
    nTimeElapsedRetract: INT; //Elapsed time while retracting cylinder
    bSolenoidActive: BOOL; //Status input of valve solenoid
    sStatus: STRING; //Pneumatic cylinder current status
    bInterlocked: BOOL; //Interlock siganl active
    bPSSPermitOK: BOOL; //Status of the PSS permit signal
    bError: BOOL; //Pneumatic axis is in Error state
END_STRUCT
END_TYPE

// ---- tc_mca_std_lib/DUTs/Pneumatics/ST_PneumaticAxisStruct.TcDUT
TYPE ST_PneumaticAxisStruct :
STRUCT
    stPneumaticAxisInputs: ST_PneumaticAxisInputs;
    stPneumaticAxisOutputs: ST_PneumaticAxisOutputs;
    stPneumaticAxisControl: ST_PneumaticAxisControl;
    stPneumaticAxisStatus: ST_PneumaticAxisStatus;
    stPneumaticAxisConfig: ST_PneumaticAxisConfig;
    ePneumaticAxisMode: E_PneumaticMode;
    ePneumaticAxisErrors: E_PneumaticAxisErrors;
END_STRUCT
END_TYPE

// ---- tc_mca_std_lib/DUTs/E_SlitPairStates.TcDUT
{attribute 'qualified_only'}
{attribute 'strict'}
TYPE E_SlitPairStates :
(
    INIT := 0,
    INIT_CLEAR_GEARING,
    INIT_GEAROUT_CHECK,
    CHECK_HOME_STATUS,
    HOME_BLADES,
    CHECK_BLADE_HOME_COMPLETE,
    HOME_GAP,
    CHECK_GAP_HOME_COMPLETE,
    GEARIN_SLITS,
    CHECK_GEARIN_SLITS_COMPLETE,
    SLITS_OPERATIONAL,
    GEAROUT_BLADES,
    CHECK_GEAROUT_COMPLETE,
    CLEAR_GAP_CALIBRATION,
    ERROR,
    ERROR_GEAROUT,
    ERROR_GEAROUT_CHECK,
    ERROR_RESET_AXES,
    ERROR_RESET_CHECK
);
END_TYPE

// ---- tc_mca_std_lib/DUTs/E_MotionFunctions.TcDUT
{attribute 'qualified_only'}
{attribute 'strict'}
TYPE E_MotionFunctions :
(
    eMoveAbsolute := 0,
    eMoveRelative := 1,
    eMoveVelocity := 3, //Continous moving at a set velocity once bExecute goes high
    eMoveModulo := 2, //Move for 360 deg rotation, see Beckhoff docs
	eSetPosition := 4,
	eLocalMoveAbsolute := 5,
	eLocalMoveRelative := 6,
	eLocalMoveVelocity := 7,

    eHome := 10, //Run the homing routine for the axis
    eWriteParameter := 50, //Writes the set value to the set parameter once bExecute goes high
    eReadParameter := 60, //Reads a single Parameter
	eWriteToggleSWLimits := 70
) := eHome; //Home is the default behaviour of the axis.
END_TYPE

// ---- tc_mca_std_lib/DUTs/Safety_Structures/ST_DeviceDualChannelInput.TcDUT
TYPE ST_DeviceDualChannelInput :
STRUCT
	//monitored device
	stSafetyDescription : ST_SafetyDescription;
	Ch1 AT %I* : BIT;
	Ch2 AT %I* : BIT;
	inError AT %I* : BOOL;
	Output AT %I* : BOOL;
END_STRUCT
END_TYPE

// ---- tc_mca_std_lib/DUTs/Safety_Structures/ST_DeviceSingleChannelInput.TcDUT
TYPE ST_DeviceSingleChannelInput :
STRUCT
	stSafetyDescription : ST_SafetyDescription;
	Output AT %I* : BOOL;
END_STRUCT
END_TYPE

// ---- tc_mca_std_lib/DUTs/Safety_Structures/ST_SafetyDescription.TcDUT
TYPE ST_SafetyDescription :
STRUCT
	sSafetyName : STRING(nMAX_SAFETY_NAME);
	eSafetyType : E_SafetyType;
	sLocation  : STRING(nMAX_LOCATION_NAME);
END_STRUCT
END_TYPE

// ---- tc_mca_std_lib/DUTs/Safety_Structures/ST_SafetyGroup.TcDUT
TYPE ST_SafetyGroup :
STRUCT
	Connected : BOOL:= FALSE; //User to set
	STATE AT %I* : USINT; //1 - run, 2 - stop, 4 - error, 5 - reset, 6 - start, 7 - stoperror, 16 - deactive, 17 - waitcommerr
	DIAG AT %I* : USINT;//0 - no error, 1 - FbErr, 2 - CommErr, 3-ModuleError 4- CMPErr, 5 - Deactive, 6 - RestartErr
END_STRUCT
END_TYPE

// ---- tc_mca_std_lib/DUTs/Safety_Structures/ST_SafetyTargetDevice.TcDUT
TYPE ST_SafetyTargetDevice :
STRUCT
	ProjectName : STRING;
	Device : STRING;
	SERIAL AT %I* : UDINT;
	CRC AT %I*: WORD;
	RUN AT %Q* : BOOL;
	Global_RUN : BOOL:= TRUE;
	ERROR_ACK AT %Q* : BOOL;
	Global_ERROR_ACK : BOOL:= TRUE;
	aSafetyGroups : ARRAY [1..10] OF ST_SafetyGroup;
	State : USINT; //summary of group mode operation
	Diag : USINT; //summary of group mode diagnostics
	State_String : STRING;
	Diag_String : STRING;
	
	
END_STRUCT
END_TYPE

// ---- tc_mca_std_lib/DUTs/ST_McStatus.TcDUT
TYPE ST_McStatus :
STRUCT
    Done: BOOL;
    Busy: BOOL;
    Active: BOOL;
    InVelocity: BOOL;
    CommandAborted: BOOL;
    Error: BOOL;
    ErrorID: UDINT;
END_STRUCT
END_TYPE

// ---- GVLs/GVL_APP.TcGVL
{attribute 'qualified_only'}
VAR_GLOBAL
END_VAR

VAR_GLOBAL CONSTANT
    nAXIS_NUM: UINT := 1;
	nAXIS_GROUPS_NUM: INT := 1;
    nPNEUMATIC_AXIS_NUM: UINT := 0;
	nSAFETY_NUM: UINT := 1;
END_VAR

// ---- GVLs/KeTop.TcGVL
{attribute 'qualified_only'}
VAR_GLOBAL 
    alive : UINT; 
    buzzer : UINT; 
    connectionBoxAddress : UINT; 
    enSwitch : UINT; 
    handWheelPosition : DINT; 
    handWheelPressed : BOOL; 
    keyCount : ARRAY [0..127] OF UINT; 
    keys : ARRAY [ 0..127] OF BOOL; 
    keySwitch : BYTE; 
    leds : ARRAY [0..15] OF BYTE ; 
    pushButton : BYTE; 
    PushButtonLed : BYTE; 
    pushSwitch : BYTE; 
    pushSwitchLed : BYTE; 
    rotSwitch : BYTE; 
    screenBrightness : UINT := 100; 
    screenTimeout : UINT; 
    selSwitch : BYTE; 
    typePlate : ARRAY [0..5] OF UINT; 
	enSwitch1 AT %I*: BOOL; 
	enSwitch2 AT %I*: BOOL; 
END_VAR

// ---- tc_mca_std_lib/GVLs/GVL.TcGVL
VAR_GLOBAL
    // Semantic version in machine-readable format.
    // Update it and commit it immediatly before setting a tag
    nVersionMajor: UINT := 2; // Major Version
    nVersionMinor: UINT := 2; // Minor Version
    nVersionPatch: UINT := 0; // Patch level
    astAxes: ARRAY [1..GVL_APP.nAXIS_NUM] OF ST_AxisStruct; //Array of ST_AxisStruct for holding axis parameters and controls
    astPneumaticAxes: ARRAY [1..GVL_APP.nPNEUMATIC_AXIS_NUM] OF ST_PneumaticAxisStruct; //Array of ST_PneumaticAxisStruct for holding pneumatic axis parameters and controls
    iAxis: UINT; //Index for for loops while going through axes
	iSafety: UINT; //Index for loops while going through safety devices
    iGroup: INT;
	iPneumaticAxis: UINT := 1; //Index for for loops while going through pneumatic axes
    fbGetCurTaskIndex: GETCURTASKINDEX;
    bLocalMode: BOOL;
	astAxesPersistent: ARRAY [1..GVL_APP.nAXIS_NUM] OF ST_AxisPersistent;
	astAxesGroup: ARRAY [1..GVL_APP.nAXIS_GROUPS_NUM] OF ST_AxisGroupStruct;
	iAxesGroupIndex : INT;
END_VAR

VAR_GLOBAL CONSTANT
    nMAX_AXIS_NAME: UINT := 32;
    nMAX_AXIS_GROUP_NAME: UINT := 32;
	nMAX_AXES_PER_GROUP: INT := 9;	nMAX_SAFETY_NAME: UINT := 32;
	nMAX_LOCATION_NAME: UINT := 32;
END_VAR

// ---- tc_mca_std_lib/GVLs/GVL_UnitStrings.TcGVL
VAR_GLOBAL CONSTANT
	UNIT_mm : STRING := 'mm';
	UNIT_degree : STRING := 'deg';
	UNIT_radians : STRING := 'rad';
END_VAR

// ---- tc_mca_std_lib/DUTs/I_Axis.TcIO
INTERFACE I_Axis

METHOD EndOfCycle : BOOL
VAR_INPUT
END_VAR
END_METHOD

METHOD Run : BOOL
VAR_INPUT
END_VAR
END_METHOD

PROPERTY stAxis : REFERENCE TO ST_AxisStruct
GET
END_GET
SET
END_SET
END_PROPERTY

END_INTERFACE

// ---- POUs/MAIN.TcPOU
PROGRAM MAIN
VAR
	run1 : BOOL;
	run2 : BOOL;

    sVersion: STRING := '1.0.0';
    aIAxes: ARRAY [1..GVL_APP.nAXIS_NUM] OF I_Axis;
    afbAxes: ARRAY [1..GVL_APP.nAXIS_NUM] OF FB_Axis;
    afbPneumaticAxes: ARRAY [1..GVL_APP.nPNEUMATIC_AXIS_NUM] OF FB_PneumaticAxis;
    hmiAxisSelection: INT := 1; //Not possible to use local hmi variables for array indexes
    hmiPneumaticAxisSelection: INT := 1;
	retainHandlerPresent : BOOL := TRUE;	//Set true if Novram present, otherwise relying on 1s UPS
	
//Startup, Shutdown and UPS
    fbUPS: FB_S_UPS_CX51x0;
    eUpsMode: E_S_UPS_Mode := eSUPS_WrPersistData_Shutdown;
    eStartUp: (eColdStart, eReadAxisFeedbackType, eCheckReadDone, eExecuteRestore, eCheckRestore, eFinishRestore);
    bAllEncRefValid : BOOL:= FALSE;
    bRestoreExecute: BOOL := FALSE;
	restoreCounter : UINT:=0;
	restoreCounterMax: UINT:=10;
    bExecuteReadEncRefSys: BOOL := FALSE;
    nRetry: INT;
    iAxes: UINT; //index for for loops in Position recovery actions
    afbReadEncRefSys: ARRAY [1..GVL_APP.nAXIS_NUM] OF MC_ReadParameter;
    afbSetPosition: ARRAY [1..GVL_APP.nAXIS_NUM] OF MC_SetPosition;
    afbReadPositionBias: ARRAY [1..GVL_APP.nAXIS_NUM] OF MC_ReadParameter;
    afbWritePositionBias: ARRAY [1..GVL_APP.nAXIS_NUM] OF MC_WriteParameter;
    fbGetDeviceIdentification: FB_GetDeviceIdentificationEx;
	
	
	
END_VAR

VAR
    bRestoreOnStartup: BOOL := TRUE;
	bPositionRestoreDone: BOOL := FALSE;
END_VAR

//POSITION_RECOVERY();


PROG();
AXES();

//IF run1 THEN
	RESTORE_POSITIONS();
//END_IF
//IF run2 THEN
	IF bPositionRestoreDone THEN
		STORE_PERSISTENT();
	END_IF
//END_IF

ACTION AXES:
//First cycle, assign FB_axis to interface array
IF _TaskInfo[fbGetCurTaskIndex.index].FirstCycle THEN
    FOR GVL.iAxis := 1 TO GVL_APP.nAXIS_NUM DO
        afbAxes[GVL.iAxis].stAxis REF= astAxes[GVL.iAxis];
        aIAxes[GVL.iAxis] := afbAxes[GVL.iAxis];
    END_FOR
    //Custom axis types defined and linked to aiAxes here
      //FB_CustomAxis extends FB_axis
        //fbCustomAxis.stAxis REF= astAxes[x];
        //aIAxes[x] := fbCustomAxis;
END_IF

//Execute FB_Axis logic
FOR GVL.iAxis := 1 TO GVL_APP.nAXIS_NUM DO
    aIAxes[GVL.iAxis].Run();
END_FOR

//Execute Pneumatic Axis logic
FOR GVL.iPneumaticAxis := 1 TO GVL_APP.nPNEUMATIC_AXIS_NUM DO
    afbPneumaticAxes[GVL.iPneumaticAxis](stPneumaticAxisStruct := GVL.astPneumaticAxes[GVL.iPneumaticAxis]);
END_FOR
END_ACTION

ACTION CHECK_UPS:
fbUPS(eUpsMode := eUpsMode);

FOR iAxes := 1 TO GVL_APP.nAXIS_NUM DO
    //Read encoder position BIAS
    IF astAxes[iAxes].stStatus.bAxisInitialized THEN
        afbReadPositionBias[iAxes](Axis := GVL.astAxes[iAxes].Axis,
                        Enable := TRUE,
                        ReadMode:= READMODE_CYCLIC,
                        ParameterNumber := E_AxisParameters.AxisEncoderOffset);
    END_IF
END_FOR

IF retainHandlerPresent AND bPositionRestoreDone THEN
	bRestoreOnStartup := TRUE;
    STORE_PERSISTENT();
    RETURN;
END_IF

IF eGlobalSUpsState = eSUPS_PowerFailure THEN
    //first cycle of powerfailure
    //execute code that should only be done once with each powerfailure, i.e. increase powerfailure counter
    bRestoreOnStartup := TRUE;
    STORE_PERSISTENT();
    RETURN;
ELSIF eGlobalSUpsState <> eSUPS_PowerOK THEN
    //next cycles of powerfailure
    //skip regular code execution for the remaining cycles of the powerfailure/writing of persistent data/quick shutdown...
    RETURN;
END_IF
END_ACTION

ACTION POSITION_RECOVERY:
fbGetDeviceIdentification(bExecute := TRUE);
IF (fbGetDeviceIdentification.stDevIdent.strHardwareSerialNo <> '') THEN
    CHECK_UPS();
    RESTORE_POSITIONS();
END_IF
END_ACTION

ACTION PROG:
//Get task index for Axes parameters initialization.
GVL.fbGetCurTaskIndex();

//Call the programs that are defined in the "Application Specific" folder.
//Create as many programs in that folder as axes and applications you have or need

//Axes initial parameters and program
//Axis_Template();
//Group_Template();
//Pneumatics_Template();

//Application program calls
//Application_Template();



Axis1();
END_ACTION

ACTION RESTORE_POSITIONS:
//This ACT will restore the position of an incremental axis on startup with the act position it read before losing power.
//It checks the type of axis, 0=incremental, and that the axis was stationary at shut down.
//Because 0 equates to incremental we also need to check that the data is valid, otherwise by default it would restore all axes.
//By default an axis will not restore the position unless it is set to opt-in, i.e. GVL.aAxes[iAxes].stConfig.eRestorePosition is non-zero.
//This needs to be initialised somewhere in TwinCAT code otherwise it will not be available at start up.
//A restore will only be performed on a loss of power, this code shouldn't make any changes on a reset cold, a rest origin or a download.
//There is a enum to allow for different types of restore modes, currently only one is implemented.
//0 'DontRestore'
//1 'RestoreWithoutHome' -restores the position using a set position fb and does not set the home bit in the axis struct.
//Note from Beckhoff: "A maximum of 1 MB persistent data can be reliably saved over the entire service life."
//Encoder Reference system types: https://infosys.beckhoff.com/english.php?content=../content/1033/tf50x0_tc3_nc_ptp/3439907723.html&id=
//INCREMENTAL=0;
//ABSOLUTE=1;
//ABSOLUTE (modulo)=2;
//ABSOLUTE MULTITURN RANGE (with single overflow)=3;
//INCREMENTAL (singleturn absolute)=4;
//ABSOLUTE SINGLETURN RANGE (with single overflow)=5;

IF NOT bPositionRestoreDone THEN
	bRestoreExecute := TRUE;
END_IF


//Upon startup bPositionRestoreDone will be set to FALSE, after successfully completing the following code it will be set TRUE
//and should stay TRUE for the rest of the time the PLC is operational, thus this routine should only be completed once.
IF bRestoreExecute AND NOT bPositionRestoreDone THEN
    //Cycle through function blocks that read the encoder reference system i.e. whether axis is incremental or absolute
    FOR iAxes := 1 TO GVL_APP.nAXIS_NUM DO
         afbReadEncRefSys[iAxes](
            Axis := GVL.astAxes[iAxes].Axis,
            ParameterNumber := MC_AxisParameter.AxisEncoderReferenceSystem,
            ReadMode := E_READMODE.READMODE_ONCE);
    END_FOR

    //Cycle through set position and MC_WritePArameter function blocks for each axis
    FOR iAxes := 1 TO GVL_APP.nAXIS_NUM DO
        afbSetPosition[iAxes](
            Axis := GVL.astAxes[iAxes].Axis,
            Position := astAxesPersistent[iAxes].fPositionAtShutdown);

        afbWritePositionBias[iAxes](
            Axis:= GVL.astAxes[iAxes].Axis,
            ParameterNumber:= E_AxisParameters.AxisEncoderOffset,
            Value:= astAxesPersistent[iAxes].fEncoderBiasAtShutdown);
    END_FOR

    CASE eStartUp OF
        eColdStart:
            //First cycle of the PLC, do nothing just give one cycle for variables to initialise
            IF NOT bPositionRestoreDone THEN
				FOR iAxes := 1 TO GVL_APP.nAXIS_NUM DO
					afbReadEncRefSys[iAxes].Enable := FALSE;                         
            	END_FOR
                eStartUp := eReadAxisFeedbackType;
                nRetry := 0;
            END_IF

        eReadAxisFeedbackType:
            //Exectute the function blocks to read the encoder reference system (0=inc OR 1=ABS)
            FOR iAxes := 1 TO GVL_APP.nAXIS_NUM DO
				
				IF NOT afbReadEncRefSys[iAxes].Valid THEN
					afbReadEncRefSys[iAxes].Enable := TRUE; 
				END_IF
					                        
            END_FOR
			eStartUp := eCheckReadDone;

        eCheckReadDone:
            //Check the encoder reference system has been read for all axis -> if busy then continue with PLC cycle and check again next time.
            //If afbReadEncRefSys not started then go back a step.
            //If any axes result in an error the code will get stuck here, this happens if GVL_APP.nAXIS_NUM is not set correctly
			bAllEncRefValid:= TRUE;
            FOR iAxes := 1 TO GVL_APP.nAXIS_NUM DO
				IF afbReadEncRefSys[iAxes].Valid THEN
					bAllEncRefValid:= bAllEncRefValid AND TRUE;
				ELSIF NOT afbReadEncRefSys[iAxes].Busy AND NOT afbReadEncRefSys[iAxes].Valid THEN
					 afbReadEncRefSys[iAxes].Enable := NOT  afbReadEncRefSys[iAxes].Enable;
					 bAllEncRefValid:= FALSE;
				ELSIF afbReadEncRefSys[iAxes].Busy THEN
					bAllEncRefValid:= FALSE;
				END_IF
                (*IF NOT afbReadEncRefSys[iAxes].Valid THEN
                    IF afbReadEncRefSys[iAxes].Busy THEN
                        //Exit MAIN.STARTUP Action and wait till next cycle, needs to cycle through whole program in order for data to update
                        RETURN;
                    ELSE
                        //Sometimes the code gets here and the afbReadEncRefSys[iAxes] misses the rising edge. If  the code gets here it means
                        //valid=FALSE and .busy=FALSE which indicateds the FB probably hasn't started and thus needs to see a rising edge.
                        //Set execute to low, Exit MAIN.STARTUP and go back a step in the CASE statement.
                        afbReadEncRefSys[iAxes].Enable := FALSE;
                        eStartUp := eReadAxisFeedbackType;
                        nRetry := nRetry + 1; //counter used for troubleshooting to see how many cycles it takes before afbReadEncRefSys function blocks are read correctly
                        RETURN;
                    END_IF
                END_IF*)
            END_FOR
            //If the code gets here all axes have .valid=TRUE for all axes
			IF bAllEncRefValid THEN
				eStartUp := eExecuteRestore;
			ELSE
				eStartUp:= eReadAxisFeedbackType;
			END_IF
            

        eExecuteRestore:
            //Execute position and encoder BIAS restore by setting Execute = TRUE
           FOR iAxes := 1 TO GVL_APP.nAXIS_NUM DO
                IF GVL.astAxes[iAxes].stConfig.eRestorePosition = E_RestorePosition.eRestoreWithoutHome THEN
                    //Restore position value for incremental encoders
                    IF afbReadEncRefSys[iAxes].Value = 1 OR
                    afbReadEncRefSys[iAxes].Value = 3 OR
                    afbReadEncRefSys[iAxes].Value = 5 THEN
                       afbWritePositionBias[iAxes].Execute := TRUE;
					ELSIF NOT astAxesPersistent[iAxes].bMovingAtShutdown THEN
                       afbSetPosition[iAxes].Execute := TRUE;
                    //Restore encoder position BIAS for absolute encoders

                    END_IF
                END_IF
            END_FOR
			restoreCounter:= restoreCounter+1;
            eStartUp := eCheckRestore;


        eCheckRestore:
            //Check the set position and write enocder BIAS fbs are finished
            //Nothing actually happens if the restore is not done, the code just returns from here each cycle and the
            //bPositionRestoreDone will never get set to TRUE and will take up cycle time
			IF restoreCounter>restoreCounterMax THEN
				eStartUp:= eFinishRestore;
				RETURN;
			END_IF
            eStartUp:= eFinishRestore;
			FOR iAxes := 1 TO GVL_APP.nAXIS_NUM DO

                IF GVL.astAxes[iAxes].stConfig.eRestorePosition = E_RestorePosition.eRestoreWithoutHome THEN
                    IF afbReadEncRefSys[iAxes].Value = 1 OR
                     afbReadEncRefSys[iAxes].Value = 3 OR
                     afbReadEncRefSys[iAxes].Value = 5 THEN
                        IF NOT afbWritePositionBias[iAxes].Done THEN
                            afbWritePositionBias[iAxes].Execute := FALSE;
                            eStartUp := eExecuteRestore;
                            RETURN;
                        END_IF
					ELSIF NOT astAxesPersistent[iAxes].bMovingAtShutdown THEN
                        IF NOT afbSetPosition[iAxes].Done THEN
                            afbSetPosition[iAxes].Execute := FALSE;
                            eStartUp := eExecuteRestore;
                            RETURN;
                        END_IF

                    END_IF
                END_IF
            END_FOR


        eFinishRestore:
            //Remove execute = TRUE for afbRestorePosition and fbWritePositionBias
            FOR iAxes := 1 TO GVL_APP.nAXIS_NUM DO
                afbSetPosition[iAxes].Execute := FALSE;
                afbWritePositionBias[iAxes].Execute := FALSE;
                bPositionRestoreDone := TRUE;
                bRestoreExecute := FALSE;
            END_FOR
    END_CASE
END_IF
END_ACTION

ACTION STORE_PERSISTENT:
FOR iAxes := 1 TO GVL_APP.nAXIS_NUM DO
    //Read encoder position BIAS
    IF astAxes[iAxes].stStatus.bAxisInitialized THEN
        afbReadPositionBias[iAxes](Axis := GVL.astAxes[iAxes].Axis,
                        Enable := TRUE,
                        ReadMode:= READMODE_CYCLIC,
                        ParameterNumber := E_AxisParameters.AxisEncoderOffset);
    END_IF
END_FOR

FOR iAxes := 1 TO GVL_APP.nAXIS_NUM DO
    //Store Position beofre shutdown
    astAxesPersistent[iAxes].fPositionAtShutdown := GVL.astAxes[iAxes].Axis.NcToPlc.ActPos;

    //Store encoder position BIAS at shutdown
	
    astAxesPersistent[iAxes].fEncoderBiasAtShutdown := afbReadPositionBias[iAxes].Value;

    //Store value of moving at shutdown
    IF GVL.astAxes[iAxes].Axis.Status.StandStill OR GVL.astAxes[iAxes].Axis.Status.Disabled THEN
        astAxesPersistent[iAxes].bMovingAtShutdown := FALSE;
    ELSE
        astAxesPersistent[iAxes].bMovingAtShutdown := TRUE;
    END_IF
END_FOR
END_ACTION

END_PROGRAM

// ---- tc_mca_std_lib/POUs/Motion/FB_Axis.TcPOU
//Function block to run a virtual drive with Nc
FUNCTION_BLOCK FB_Axis IMPLEMENTS I_axis
VAR
    _stAxis: REFERENCE TO ST_AxisStruct; // Local property pointer for axis structure
    astMcStatus: ARRAY[1..nMCSTATUS_ARRAY_SIZE] OF POINTER TO ST_McStatus; //Array of all MC status signals defined in FB_init

    fbPower: MC_Power;
    stMcStatusPower: ST_McStatus;

    fbStop: MC_Stop;
    stMcStatusStop: ST_McStatus;

    fbHalt: MC_Halt;
    stMcStatusHalt: ST_McStatus;

    fbReset: MC_Reset;
    stMcStatusReset: ST_McStatus;

    fbMoveAbsolute: MC_MoveAbsolute;
    fbMoveAbsolute2: MC_MoveAbsolute;
    stMcStatusMoveAbsolute: ST_McStatus;
	
	fbLocalMoveAbsolute: MC_MoveAbsolute;
    fbLocalMoveAbsolute2: MC_MoveAbsolute;
    stMcStatusLocalMoveAbsolute: ST_McStatus;

    fbMoveRelative: MC_MoveRelative;
    stMcStatusMoveRelative: ST_McStatus;
	
	fbLocalMoveRelative: MC_MoveRelative;
    stMcStatusLocalMoveRelative: ST_McStatus;

    fbMoveVelocity: MC_MoveVelocity;
    stMcStatusMoveVelocity: ST_McStatus;
	
	fbLocalMoveVelocity: MC_MoveVelocity;
    stMcStatusLocalMoveVelocity: ST_McStatus;

    fbMoveModulo: MC_MoveModulo;
    fbMoveModulo2: MC_MoveModulo;
    stMcStatusMoveModulo: ST_McStatus;
	
	fbEnableSPG : MC_ExtSetPointGenEnable;
	stMcStatusEnableSPG : ST_McStatus;
	fbDisableSPG : MC_ExtSetPointGenDisable;
	stMcStatusDisableSPG : ST_McStatus;
	

    fbHome: FB_Homing;
    stMcStatusHome: ST_McStatus;

    fbReadParameter: MC_ReadParameter;
    stMcStatusReadParameter: ST_McStatus;

    fbWriteParameter: MC_WriteParameter;
    stMcStatusWriteParameter: ST_McStatus;
	fbWriteSWLimitMax: MC_WriteBoolParameter;
	fbWriteSWLimitMin: MC_WriteBoolParameter;
	stMcStatusWriteSWLimits : ST_McStatus;

	
	fbSetPosition: MC_SetPosition;
	stMcStatusSetPosition: ST_McStatus;

    //Variables for holding limits during homing
    bWaitForStopAfterLimitHit: BOOL := FALSE;
    fbRemovePowerTimer: TOF;

    //Dedicated NC parameter read FBs
    fbReadAxisVeloManSlow: MC_ReadParameter;
    fbReadAxisVeloManFast: MC_ReadParameter;
    fbReadHomingVelToCam: MC_ReadParameter;
    fbReadHomingVelFromCam: MC_ReadParameter;
    fbReadAxisVeloMax: MC_ReadParameter;
    fbReadAxisMaxAcc: MC_ReadParameter;
    fbReadAxisMaxDec: MC_ReadParameter;
    fbReadAxisAcc: MC_ReadParameter;
    fbReadAxisDec: MC_ReadParameter;
    fbReadEnMinSoftPosLimit: MC_ReadParameter;
    fbReadEnMaxSoftPosLimit: MC_ReadParameter;
    fbReadMinSoftPosLimit: MC_ReadParameter;
    fbReadMaxSoftPosLimit: MC_ReadParameter;
    fbReadEnPositionLagMonitoring: MC_ReadParameter;
    fbReadAxisMaxPosLagValue: MC_ReadParameter;
    fbReadEnTargetPositionMonitoring: MC_ReadParameter;
    fbReadTargetPositionWindow: MC_ReadParameter;

    //Edge detection triggers for statuses
    fbDoneRTrig: R_TRIG;
    fbErrorRTrig: R_TRIG;
    fbCommandAbortedRTrig: R_TRIG;
    fbInVelocityRTrig: R_TRIG;
    fbInVelocityFTrig: F_TRIG;
    fbExecuteRTrig: R_TRIG;
    fbStopFinishedRiseEdge: R_TRIG;
    fbHaltFinishedRiseEdge: R_TRIG;
    fbResetFinishedRiseEdge: R_TRIG;
    fbAbsMovDyn1RiseEdge: R_TRIG;
    fbAbsMovDyn2RiseEdge: R_TRIG;
	fbLocalAbsMovDyn1RiseEdge: R_TRIG;
    fbLocalAbsMovDyn2RiseEdge: R_TRIG;
    fbModMovDyn1RiseEdge: R_TRIG;
    fbModMovDyn2RiseEdge: R_TRIG;
	
	fbMoveInProgressFTrig : F_TRIG;
	fbMoveInProgressEndTimer : TON;
	fbNewMoveRTrig : R_TRIG;
	bStartOfMove : BOOL;
	bEndOfMove : BOOL;
	
	fbBwdLimitFTrig : F_TRIG;
	fbFwdLimitFTrig : F_TRIG;
	
	bSpgEnableReq : BOOL;
	bSpgDisableReq : BOOL;
	spgDisableCommand : BOOL;

	iNameCharacterIndex : int;
END_VAR
VAR CONSTANT
    nRATIO_DENOMINATOR_DEFAULT: UINT := 1;
    nNO_GEARING: UINT := 0;
    nMCSTATUS_ARRAY_SIZE: UINT := 13;
    nMULTI_MASTER_MAX_AXES: UINT := 4;
END_VAR

METHOD EndOfCycle : BOOL

_stAxis.stControl.bExecute := FALSE;
END_METHOD

METHOD FB_init : BOOL
VAR_INPUT
    bInitRetains: BOOL; // if TRUE, the retain variables are initialized (warm start / cold start)
    bInCopyCode: BOOL; // if TRUE, the instance afterwards gets moved into the copy code (online change)
END_VAR

//Copy address locations for statuses to an array to allow for easier checking of statuses
astMcStatus[1] := ADR(stMcStatusPower);
astMcStatus[2] := ADR(stMcStatusStop);
astMcStatus[3] := ADR(stMcStatusHalt);
astMcStatus[4] := ADR(stMcStatusReset);
astMcStatus[5] := ADR(stMcStatusMoveAbsolute);
astMcStatus[6] := ADR(stMcStatusMoveRelative);
astMcStatus[7] := ADR(stMcStatusMoveVelocity);
astMcStatus[8] := ADR(stMcStatusMoveModulo);
astMcStatus[9] := ADR(stMcStatusHome);
astMcStatus[10] := ADR(stMcStatusSetPosition);
astMcStatus[11] := ADR(stMcStatusReadParameter);
astMcStatus[12] := ADR(stMcStatusWriteParameter);
astMcStatus[13] := ADR(stMcStatusWriteSWLimits);
END_METHOD

METHOD mControl_AutoEnableDisable : BOOL
VAR_INPUT
END_VAR
//Has a move been requested?
IF (_stAxis.stControl.eCommand = E_MotionFunctions.eMoveAbsolute AND _stAxis.stInputs.bAllowRemoteControl) OR 
	(_stAxis.stControl.eCommand = E_MotionFunctions.eMoveModulo AND _stAxis.stInputs.bAllowRemoteControl) OR
	(_stAxis.stControl.eCommand = E_MotionFunctions.eMoveRelative AND _stAxis.stInputs.bAllowRemoteControl) OR
	(_stAxis.stControl.eCommand = E_MotionFunctions.eMoveVelocity AND _stAxis.stInputs.bAllowRemoteControl) OR
	(_stAxis.stControl.eCommand = E_MotionFunctions.eHome AND _stAxis.stInputs.bAllowRemoteControl) OR
	(_stAxis.stControl.eCommand = E_MotionFunctions.eLocalMoveAbsolute AND NOT _stAxis.stInputs.bAllowRemoteControl) OR
	(_stAxis.stControl.eCommand = E_MotionFunctions.eLocalMoveRelative AND NOT _stAxis.stInputs.bAllowRemoteControl) OR
	(_stAxis.stControl.eCommand = E_MotionFunctions.eLocalMoveVelocity AND NOT _stAxis.stInputs.bAllowRemoteControl) THEN
	IF _stAxis.stControl.bExecute AND _stAxis.stStatus.bMoveRequested = FALSE AND _stAxis.stInputs.bPermit THEN
		//new logic here to stop commands queuing with axes disabled if not meant to autoenable/disable
 		IF _stAxis.stStatus.bEnabled = FALSE AND _stAxis.stControl.bAutoEnableDisable = FALSE THEN
			_stAxis.stStatus.bMoveRequested := FALSE;
		ELSE
			_stAxis.stStatus.bMoveRequested := TRUE;
		END_IF
		//_stAxis.stStatus.bMoveRequested := TRUE;
	END_IF
ELSIF _stAxis.stControl.bExecute THEN
	ADSLOGSTR(
		msgCtrlMask := ADSLOG_MSGTYPE_ERROR,
		msgFmtStr := 'To move you must set stInputs.bAllowRemoteControl to the opposite of %s',
		strArg := BOOL_TO_STRING(_stAxis.stInputs.bAllowRemoteControl)
	);	
END_IF

IF _stAxis.stControl.bOverrideReadyToMove THEN
	_stAxis.stStatus.bReadyToMove := _stAxis.stControl.bExtReadyToMove;
ELSE
	_stAxis.stStatus.bReadyToMove := _stAxis.stStatus.bEnabled;
END_IF

//prevent the turn off if homing
IF fbMoveInProgressFTrig.Q AND NOT _stAxis.stStatus.bInHomingSeq THEN
	//start end move timer
	bEndOfMove:= TRUE;
	_stAxis.stControl.bExtReadyToMove:= FALSE;
END_IF
IF bStartOfMove THEN
	bEndOfMove:= FALSE;
	bStartOfMove:= FALSE;
END_IF

fbMoveInProgressEndTimer(IN:= bEndOfMove,PT:= _stAxis.stControl.tMoveFinishedDelay);

//If we want autoenabledisable
IF _stAxis.stControl.bAutoEnableDisable THEN
	//and a move has been requested and we are not enabled
	IF _stAxis.stStatus.bMoveRequested AND NOT _stAxis.stControl.bWaitBeforeEnable THEN
		IF _stAxis.stStatus.bMoveRequested AND _stAxis.stStatus.bEnabled = FALSE THEN
			_stAxis.stControl.bEnable:= TRUE;
		END_IF
	ELSIF _stAxis.stStatus.bMoveRequested AND _stAxis.stControl.bWaitBeforeEnable AND _stAxis.stStatus.bEnabled = FALSE AND _stAxis.stControl.bReadyToEnable THEN
		_stAxis.stControl.bEnable:= TRUE;
		_stAxis.stControl.bReadyToEnable:= FALSE;
	END_IF
	
	
	IF _stAxis.stStatus.bMoveRequested = FALSE AND fbMoveInProgressEndTimer.Q THEN
	_stAxis.stControl.bEnable:= FALSE;
	bEndOfMove := FALSE;
	END_IF
END_IF

IF _stAxis.Axis.Status.Moving THEN
	_stAxis.stStatus.bMoveInProgress := TRUE;
END_IF

IF _stAxis.Axis.Status.NotMoving AND (_stAxis.Axis.Status.InTargetPosition OR NOT _stAxis.stInputs.bLimitBwd OR NOT _stAxis.stInputs.bLimitFwd) THEN
	_stAxis.stStatus.bMoveInProgress := FALSE;
END_IF

fbNewMoveRTrig(CLK:= _stAxis.stStatus.bMoveInProgress);
IF fbNewMoveRTrig.Q THEN
	bStartOfMove:= TRUE;
END_IF
fbMoveInProgressFTrig(CLK:= _stAxis.stStatus.bMoveInProgress OR spgDisableCommand);
//No move requested and no move in progress
END_METHOD

METHOD mControl_DisableSPG : BOOL
VAR_INPUT
END_VAR
IF _stAxis.stSpg.DisableSPG THEN
	//fbEnableSPG.Execute := TRUE;
	bSpgDisableReq := TRUE;
END_IF

IF _stAxis.stStatus.bEnabled = FALSE AND bSpgDisableReq THEN
	_stAxis.stStatus.messageString:= 'Axis is disabled';
	bSpgDisableReq:= FALSE;
END_IF

IF _stAxis.stStatus.SPGEnabled = FALSE AND bSpgDisableReq THEN
	stAxis.stStatus.messageString:= 'Axis is not in ExtSPG mode';
	bSpgDisableReq:= FALSE;
END_IF





fbDisableSPG.Execute:= bSpgDisableReq;
fbDisableSPG(Axis:= _stAxis.Axis);
IF _stAxis.stControl.bAutoEnableDisable THEN
	spgDisableCommand := fbDisableSPG.Done;
END_IF

_stAxis.stSpg.DisableSPG:= FALSE;
fbDisableSPG.Execute := FALSE;
END_METHOD

METHOD mControl_EnableSPG : BOOL
VAR_INPUT
END_VAR
IF _stAxis.stSpg.EnableSPG THEN
	//fbEnableSPG.Execute := TRUE;
	bSpgEnableReq := TRUE;
END_IF

IF _stAxis.stControl.bAutoEnableDisable = FALSE AND _stAxis.stStatus.bEnabled = FALSE AND bSpgEnableReq THEN
	_stAxis.stStatus.messageString:= 'Axis must be enabled before enabling ExtSPG';
	bSpgEnableReq:= FALSE;
END_IF

IF _stAxis.stControl.bAutoEnableDisable  AND _stAxis.stStatus.bEnabled = FALSE AND bSpgEnableReq = TRUE THEN
	_stAxis.stControl.bEnable:= TRUE;
END_IF


IF _stAxis.stStatus.bEnabled THEN
	fbEnableSPG.Execute := bSpgEnableReq;
	bSpgEnableReq := FALSE;
END_IF

fbEnableSPG(Axis:= _stAxis.Axis);

_stAxis.stSpg.EnableSPG:= FALSE;
fbEnableSPG.Execute := FALSE;
END_METHOD

METHOD mControl_FeedSPG : BOOL
VAR_INPUT
END_VAR

VAR
	DirectionInternal : DINT;
END_VAR
(* 
Direction 1 = Forward
Direction -1 = Backward
Direction 0 = Standstill
*)

IF _stAxis.stSpg.OverrideDirection THEN
	DirectionInternal:= _stAxis.stSpg.Direction;
ELSE
	//Direction calculation logic
	IF _stAxis.stSpg.Velocity > ABS(_stAxis.stSpg.VelocityStandstillThreshold) THEN
		DirectionInternal := 1;
	ELSIF _stAxis.stSpg.Velocity < -ABS(_stAxis.stSpg.VelocityStandstillThreshold) THEN
		DirectionInternal := -1;
	ELSE
		DirectionInternal := 0;
	END_IF
END_IF

MC_ExtSetPointGenFeed(
	Axis:= _stAxis.Axis, 
	Position:= _stAxis.stSpg.Position,
	Velocity:= _stAxis.stSpg.Velocity,
	Acceleration:= _stAxis.stSpg.Acceleration,
	Direction:= _stAxis.stSpg.Direction);
END_METHOD

METHOD mControl_Home : ST_McStatus
IF _stAxis.stHomingConfig.eHomeSeq = E_HomingRoutines.eNoHoming THEN
    _stAxis.stStatus.bHomed := TRUE;
END_IF

IF _stAxis.stControl.eCommand = E_MotionFunctions.eHome THEN
    //fbHome.bExecute := _stAxis.stControl.bExecute;
	IF _stAxis.stStatus.bReadyToMove THEN
		fbHome.bExecute := _stAxis.stStatus.bMoveRequested;
		IF _stAxis.stStatus.bMoveRequested THEN
			_stAxis.stStatus.bMoveRequested := FALSE;
		END_IF
	END_IF
END_IF


fbHome.eHomeSeq := _stAxis.stHomingConfig.eHomeSeq;
fbHome.fHomePosition := _stAxis.stHomingConfig.fHomePosition;
fbHome.fHomeFinishDistance := _stAxis.stHomingConfig.fHomeFinishDistance;
fbHome.fHomeAbsPosition:= _stAxis.stHomingConfig.fHomeAbsPosition;
fbHome.fHomeMidRelativeMove := _stAxis.stHomingConfig.fHomeMidRelativeMove;
fbHome.bGoToBwdLimitFirst:= _stAxis.stHomingConfig.bGoToBwdFirst;
fbHome.bGoToFwdLimitFirst:= _stAxis.stHomingConfig.bGoToFwdFirst;
fbHome.fFastVelocity:= _stAxis.stControl.fVelocity;
fbHome.bDoAbsoluteMove:= _stAxis.stHomingConfig.bDoAbsoluteMoveAtEnd;

fbHome(
	AxisRef:= _stAxis.Axis,
    bLimitBwd := _stAxis.stInputs.bLimitBwd,
    bLimitFwd := _stAxis.stInputs.bLimitFwd,
    bHomeSensor := _stAxis.stInputs.bHomeSensor,
    stConfig := _stAxis.stConfig);
fbHome.bExecute := FALSE;
_stAxis.stStatus.bInHomingSeq:= fbHome.bInHomingSequence;

mControl_Home.Busy := fbHome.bBusy;
mControl_Home.CommandAborted := fbHome.bCommandAborted;
mControl_Home.Done := fbHome.bDone;
mControl_Home.Error := fbHome.bError;
mControl_Home.ErrorID := fbHome.nErrorId;

IF fbHome.bError THEN
    _stAxis.stError.nHomeErrorID := fbHome.nErrorID; //Set the error
END_IF
END_METHOD

METHOD mControl_LimitEdge : BOOL
VAR_INPUT
END_VAR
IF NOT _stAxis.Axis.Status.Homing THEN
	fbBwdLimitFTrig(CLK:= _stAxis.stInputs.bLimitBwd);
	fbFwdLimitFTrig(CLK:= _stAxis.stInputs.bLimitFwd);
END_IF

IF fbBwdLimitFTrig.Q OR fbFwdLimitFTrig.Q THEN
	_stAxis.stControl.bReset:= TRUE;
END_IF
END_METHOD

METHOD mControl_LimitHitTimer : BOOL

//Timer for keeping power on after limit switch hit, needed for homing routines - if power is lost routines are aborted
fbRemovePowerTimer(IN := _stAxis.stInputs.bLimitFwd AND _stAxis.stInputs.bLimitBwd, PT := T#100MS);

IF stMcStatusHome.Busy AND (fbRemovePowerTimer.Q OR _stAxis.Axis.NcToPlc.AxisState = 5) THEN //5=PHASE_ACCNEG
    bWaitForStopAfterLimitHit := TRUE;
ELSE
    bWaitForStopAfterLimitHit := FALSE;
END_IF
END_METHOD

METHOD mControl_LimitLinking : BOOL

_stAxis.stStatus.bFwEnabled := _stAxis.stInputs.bLimitFwd OR _stAxis.stControl.bOverrideLimits; 
_stAxis.stStatus.bBwEnabled := _stAxis.stInputs.bLimitBwd OR _stAxis.stControl.bOverrideLimits;
_stAxis.stStatus.bInterlockedFwd := _stAxis.stControl.bInterlockFwd;
_stAxis.stStatus.bInterlockedBwd := _stAxis.stControl.bInterlockBwd;
END_METHOD

METHOD mControl_Power : ST_McStatus
fbPower.Enable := _stAxis.stControl.bEnable;
IF _stAxis.Commissioning THEN
	_stAxis.stControl.bInterlockFwd:= NOT(_stAxis.stStatus.bBwEnabled AND _stAxis.stStatus.bFwEnabled);
	_stAxis.stControl.bInterlockBwd:= NOT(_stAxis.stStatus.bBwEnabled AND _stAxis.stStatus.bFwEnabled);
END_IF

fbPower.Enable_Negative := (_stAxis.stStatus.bBwEnabled OR bWaitForStopAfterLimitHit) AND NOT _stAxis.stStatus.bInterlockedBwd;
fbPower.Enable_Positive := (_stAxis.stStatus.bFwEnabled OR bWaitForStopAfterLimitHit) AND NOT _stAxis.stStatus.bInterlockedFwd;
fbPower.Override := _stAxis.stConfig.fOverride;

fbPower(Axis := _stAxis.Axis);

mControl_Power.Error := fbPower.Error;

IF fbPower.Error THEN
    _stAxis.stError.nPowerErrorID := fbPower.ErrorID; //Set the error
END_IF
END_METHOD

METHOD mControl_Reset : ST_McStatus
VAR
    i: UINT;
END_VAR
fbReset.Execute := _stAxis.stControl.bReset;

fbReset(Axis := _stAxis.Axis);
IF fbReset.Done THEN
    _stAxis.stStatus.bError := FALSE;
	_stAxis.stStatus.bMcError := FALSE;
    FOR i := 1 TO nMCSTATUS_ARRAY_SIZE DO
        //Clear all the errors
        _stAxis.stStatus.nErrorID := 0;
    END_FOR
	_stAxis.stStatus.nMcErrorID := 0;
END_IF

mControl_Reset.Busy := fbReset.Busy;
mControl_Reset.Done := fbReset.Done;
mControl_Reset.Error := fbReset.Error;
mControl_Reset.ErrorID := fbReset.ErrorID;

IF fbReset.Error THEN
    _stAxis.stError.nResetErrorID := fbReset.ErrorID; //Set the error
END_IF

fbResetFinishedRiseEdge(CLK:=fbReset.Done OR fbReset.Error);
IF fbResetFinishedRiseEdge.Q OR fbReset.Done THEN
    _stAxis.stControl.bReset := FALSE;
END_IF
END_METHOD

METHOD mLocalMove_MoveAbsolute : ST_McStatus
IF _stAxis.stControl.eCommand = E_MotionFunctions.eLocalMoveAbsolute THEN
	IF _stAxis.stStatus.bReadyToMove THEN
		fbLocalMoveAbsolute.Execute := _stAxis.stStatus.bMoveRequested;
		IF _stAxis.stStatus.bMoveRequested THEN
			_stAxis.stStatus.bMoveRequested := FALSE;
		END_IF
    	IF fbLocalMoveAbsolute.Execute AND fbMoveAbsolute.Busy THEN
        	fbLocalMoveAbsolute2.Execute := TRUE;
    	END_IF
	END_IF    
END_IF

// Parameters
fbLocalMoveAbsolute.Position := _stAxis.stControl.fPosition;
fbLocalMoveAbsolute.Velocity := ABS(_stAxis.stControl.fVelocity);
fbLocalMoveAbsolute.Acceleration := _stAxis.stControl.fAcceleration;
fbLocalMoveAbsolute.Deceleration := _stAxis.stControl.fDeceleration;

fbLocalMoveAbsolute2.Position := _stAxis.stControl.fPosition;
fbLocalMoveAbsolute2.Velocity := ABS(_stAxis.stControl.fVelocity);
fbLocalMoveAbsolute2.Acceleration := _stAxis.stControl.fAcceleration;
fbLocalMoveAbsolute2.Deceleration := _stAxis.stControl.fDeceleration;


// Call both move absolute FB
fbLocalMoveAbsolute(Axis := _stAxis.Axis);
fbLocalMoveAbsolute2(Axis := _stAxis.Axis);

//Reset Execute bits
fbLocalMoveAbsolute.Execute := FALSE;
fbLocalMoveAbsolute2.Execute := FALSE;


// STATUS bits
mLocalMove_MoveAbsolute.Active := fbLocalMoveAbsolute.Active OR fbLocalMoveAbsolute2.Active;
mLocalMove_MoveAbsolute.Done := fbLocalMoveAbsolute.Done OR fbLocalMoveAbsolute2.Done;
mLocalMove_MoveAbsolute.Busy := fbLocalMoveAbsolute.Busy OR fbLocalMoveAbsolute2.Busy;
mLocalMove_MoveAbsolute.Error := fbLocalMoveAbsolute.Error OR fbLocalMoveAbsolute2.Error;


// Capture the CommandAborted for first scan if the other absolute move overtakes the current
fbLocalAbsMovDyn1RiseEdge(CLK:= fbLocalMoveAbsolute.Busy AND fbLocalMoveAbsolute2.CommandAborted, Q=>);
fbLocalAbsMovDyn2RiseEdge(CLK:= fbLocalMoveAbsolute2.Busy AND fbLocalMoveAbsolute.CommandAborted, Q=>);
mLocalMove_MoveAbsolute.CommandAborted := (fbLocalMoveAbsolute.CommandAborted AND NOT fbLocalAbsMovDyn2RiseEdge.Q)
                                    OR (fbLocalMoveAbsolute2.CommandAborted AND NOT fbLocalAbsMovDyn1RiseEdge.Q);

// Error IDs
IF fbLocalMoveAbsolute.Error THEN
    _stAxis.stError.nLocalMoveAbsoluteErrorID := fbLocalMoveAbsolute.ErrorID; //Set the error
    mLocalMove_MoveAbsolute.ErrorID := fbLocalMoveAbsolute.ErrorID;
END_IF
IF fbLocalMoveAbsolute2.Error THEN
    _stAxis.stError.nLocalMoveAbsoluteErrorID := fbLocalMoveAbsolute2.ErrorID; //Set the error
    mLocalMove_MoveAbsolute.ErrorID := fbLocalMoveAbsolute2.ErrorID;
END_IF
END_METHOD

METHOD mLocalMove_MoveRelative : ST_McStatus

IF _stAxis.stControl.eCommand = E_MotionFunctions.eLocalMoveRelative THEN
	IF _stAxis.stStatus.bReadyToMove THEN
		fbLocalMoveRelative.Execute := _stAxis.stStatus.bMoveRequested;
		IF _stAxis.stStatus.bMoveRequested THEN
			_stAxis.stStatus.bMoveRequested := FALSE;
		END_IF
	END_IF
END_IF

fbLocalMoveRelative.Distance := _stAxis.stControl.fRelativePosition;
fbLocalMoveRelative.Velocity := ABS(_stAxis.stControl.fVelocity);
fbLocalMoveRelative.Acceleration := _stAxis.stControl.fAcceleration;
fbLocalMoveRelative.Deceleration := _stAxis.stControl.fDeceleration;

fbLocalMoveRelative(Axis := _stAxis.Axis);
fbLocalMoveRelative.Execute := FALSE;

mLocalMove_MoveRelative.Active := fbLocalMoveRelative.Active;
mLocalMove_MoveRelative.Done := fbLocalMoveRelative.Done;
mLocalMove_MoveRelative.Busy := fbLocalMoveRelative.Busy;
mLocalMove_MoveRelative.Error := fbLocalMoveRelative.Error;
mLocalMove_MoveRelative.ErrorID := fbLocalMoveRelative.ErrorID;
mLocalMove_MoveRelative.CommandAborted := fbLocalMoveRelative.CommandAborted;

IF fbLocalMoveRelative.Error THEN
    _stAxis.stError.nLocalMoveRelativeErrorID := fbLocalMoveRelative.ErrorID; //Set the error
END_IF
END_METHOD

METHOD mLocalMove_MoveVelocity : ST_McStatus
IF _stAxis.stControl.eCommand = E_MotionFunctions.eLocalMoveVelocity THEN
	IF _stAxis.stStatus.bReadyToMove THEN
		fbLocalMoveVelocity.Execute := _stAxis.stStatus.bMoveRequested;
		IF _stAxis.stStatus.bMoveRequested THEN
			_stAxis.stStatus.bMoveRequested := FALSE;
		END_IF
	END_IF
END_IF

fbLocalMoveVelocity.Direction := SEL(_stAxis.stControl.fVelocity < 0, MC_Positive_Direction, MC_Negative_Direction);
fbLocalMoveVelocity.Velocity := ABS(_stAxis.stControl.fVelocity);

IF fbLocalMoveVelocity.Execute THEN
	_stAxis.stControl.fVelocity := ABS(_stAxis.stControl.fVelocity);
END_IF

fbLocalMoveVelocity.Acceleration := _stAxis.stControl.fAcceleration;
fbLocalMoveVelocity.Deceleration := _stAxis.stControl.fDeceleration;

fbLocalMoveVelocity(Axis := _stAxis.Axis);
fbLocalMoveVelocity.Execute:= FALSE;

mLocalMove_MoveVelocity.Active := fbLocalMoveVelocity.Active;
mLocalMove_MoveVelocity.InVelocity := fbLocalMoveVelocity.InVelocity;
mLocalMove_MoveVelocity.Busy := fbLocalMoveVelocity.Busy;
mLocalMove_MoveVelocity.Error := fbLocalMoveVelocity.Error;
mLocalMove_MoveVelocity.ErrorID := fbLocalMoveVelocity.ErrorID;
mLocalMove_MoveVelocity.CommandAborted := fbLocalMoveVelocity.CommandAborted;

IF fbLocalMoveVelocity.Error THEN
    _stAxis.stError.nLocalMoveVelocityErrorID := fbLocalMoveVelocity.ErrorID; //Set the error
END_IF
END_METHOD

METHOD mMove_Halt : ST_McStatus
fbHalt.Deceleration := _stAxis.stControl.fDeceleration;
fbHalt.Execute := _stAxis.stControl.bHalt;

fbHalt(Axis := _stAxis.Axis);

mMove_Halt.Busy := fbHalt.Busy;
mMove_Halt.Done := fbHalt.Done;
mMove_Halt.Error := fbHalt.Error;
mMove_Halt.ErrorID := fbHalt.ErrorID;
mMove_Halt.Active := fbHalt.Active;
mMove_Halt.CommandAborted := fbHalt.CommandAborted;

IF fbHalt.Error THEN
    _stAxis.stError.nHaltErrorID := fbHalt.ErrorID; //Set the error
END_IF

//Execution of fbHalt ended
fbHaltFinishedRiseEdge(CLK:=fbHalt.Done OR fbHalt.Error OR fbHalt.CommandAborted);
IF fbHaltFinishedRiseEdge.Q OR fbHalt.Done OR fbHalt.CommandAborted THEN
    _stAxis.stControl.bHalt := FALSE;
END_IF
END_METHOD

METHOD mMove_MoveAbsolute : ST_McStatus
IF _stAxis.stControl.eCommand = E_MotionFunctions.eMoveAbsolute THEN
	IF _stAxis.stStatus.bReadyToMove THEN
		fbMoveAbsolute.Execute := _stAxis.stStatus.bMoveRequested;
		IF _stAxis.stStatus.bMoveRequested THEN
			_stAxis.stStatus.bMoveRequested := FALSE;
		END_IF
    	IF fbMoveAbsolute.Execute AND fbMoveAbsolute.Busy THEN
        	fbMoveAbsolute2.Execute := TRUE;
    	END_IF
	END_IF    
END_IF

// Parameters
fbMoveAbsolute.Position := _stAxis.stControl.fPosition;
fbMoveAbsolute.Velocity := ABS(_stAxis.stControl.fVelocity);
fbMoveAbsolute.Acceleration := _stAxis.stControl.fAcceleration;
fbMoveAbsolute.Deceleration := _stAxis.stControl.fDeceleration;

fbMoveAbsolute2.Position := _stAxis.stControl.fPosition;
fbMoveAbsolute2.Velocity := ABS(_stAxis.stControl.fVelocity);
fbMoveAbsolute2.Acceleration := _stAxis.stControl.fAcceleration;
fbMoveAbsolute2.Deceleration := _stAxis.stControl.fDeceleration;


// Call both move absolute FB
fbMoveAbsolute(Axis := _stAxis.Axis);
fbMoveAbsolute2(Axis := _stAxis.Axis);

//Reset Execute bits
fbMoveAbsolute.Execute := FALSE;
fbMoveAbsolute2.Execute := FALSE;


// STATUS bits
mMove_MoveAbsolute.Active := fbMoveAbsolute.Active OR fbMoveAbsolute2.Active;
mMove_MoveAbsolute.Done := fbMoveAbsolute.Done OR fbMoveAbsolute2.Done;
mMove_MoveAbsolute.Busy := fbMoveAbsolute.Busy OR fbMoveAbsolute2.Busy;
mMove_MoveAbsolute.Error := fbMoveAbsolute.Error OR fbMoveAbsolute2.Error;


// Capture the CommandAborted for first scan if the other absolute move overtakes the current
fbAbsMovDyn1RiseEdge(CLK:= fbMoveAbsolute.Busy AND fbMoveAbsolute2.CommandAborted, Q=>);
fbAbsMovDyn2RiseEdge(CLK:= fbMoveAbsolute2.Busy AND fbMoveAbsolute.CommandAborted, Q=>);
mMove_MoveAbsolute.CommandAborted := (fbMoveAbsolute.CommandAborted AND NOT fbAbsMovDyn2RiseEdge.Q)
                                    OR (fbMoveAbsolute2.CommandAborted AND NOT fbAbsMovDyn1RiseEdge.Q);

// Error IDs
IF fbMoveAbsolute.Error THEN
    _stAxis.stError.nMoveAbsoluteErrorID := fbMoveAbsolute.ErrorID; //Set the error
    mMove_MoveAbsolute.ErrorID := fbMoveAbsolute.ErrorID;
END_IF
IF fbMoveAbsolute2.Error THEN
    _stAxis.stError.nMoveAbsoluteErrorID := fbMoveAbsolute2.ErrorID; //Set the error
    mMove_MoveAbsolute.ErrorID := fbMoveAbsolute2.ErrorID;
END_IF
END_METHOD

METHOD mMove_MoveModulo : ST_McStatus
IF _stAxis.stControl.eCommand = E_MotionFunctions.eMoveModulo THEN
	IF _stAxis.stStatus.bReadyToMove THEN
		fbMoveModulo.Execute := _stAxis.stStatus.bMoveRequested;
		IF _stAxis.stStatus.bMoveRequested THEN
			_stAxis.stStatus.bMoveRequested := FALSE;
		END_IF
    	IF fbMoveModulo.Execute AND fbMoveAbsolute.Busy THEN
        	fbMoveModulo2.Execute := TRUE;
    	END_IF
	END_IF    
END_IF

// Parameters
fbMoveModulo.Position := _stAxis.stControl.fPosition;
fbMoveModulo.Velocity := ABS(_stAxis.stControl.fVelocity);
fbMoveModulo.Acceleration := _stAxis.stControl.fAcceleration;
fbMoveModulo.Deceleration := _stAxis.stControl.fDeceleration;

fbMoveModulo2.Position := _stAxis.stControl.fPosition;
fbMoveModulo2.Velocity := ABS(_stAxis.stControl.fVelocity);
fbMoveModulo2.Acceleration := _stAxis.stControl.fAcceleration;
fbMoveModulo2.Deceleration := _stAxis.stControl.fDeceleration;

// Call both move absolute FB
fbMoveModulo(Axis := _stAxis.Axis);
fbMoveModulo.Execute := FALSE;
fbMoveModulo2(Axis := _stAxis.Axis);
fbMoveModulo2.Execute := FALSE;

// Status bits
mMove_MoveModulo.Active := fbMoveModulo.Active OR fbMoveModulo2.Active;
mMove_MoveModulo.Done := fbMoveModulo.Done OR fbMoveModulo2.Done;
mMove_MoveModulo.Busy := fbMoveModulo.Busy OR fbMoveModulo2.Busy;
mMove_MoveModulo.Error := fbMoveModulo.Error OR fbMoveModulo2.Error;

// Capture the CommandAborted for first scan if the other absolute move overtakes the current
fbModMovDyn1RiseEdge(CLK:= fbMoveModulo.Busy AND fbMoveModulo2.CommandAborted, Q=>);
fbModMovDyn2RiseEdge(CLK:= fbMoveModulo2.Busy AND fbMoveModulo.CommandAborted, Q=>);
mMove_MoveModulo.CommandAborted := (fbMoveModulo.CommandAborted AND NOT fbModMovDyn2RiseEdge.Q)
                                    OR (fbMoveModulo2.CommandAborted AND NOT fbModMovDyn1RiseEdge.Q);

// Error IDs
IF fbMoveModulo.Error THEN
    _stAxis.stError.nMoveModuloErrorID := fbMoveModulo.ErrorID; //Set the error
    mMove_MoveModulo.ErrorID := fbMoveModulo.ErrorID;
END_IF

IF fbMoveModulo2.Error THEN
    _stAxis.stError.nMoveModuloErrorID := fbMoveModulo2.ErrorID; //Set the error
    mMove_MoveModulo.ErrorID := fbMoveModulo2.ErrorID;
END_IF
END_METHOD

METHOD mMove_MoveRelative : ST_McStatus

IF _stAxis.stControl.eCommand = E_MotionFunctions.eMoveRelative THEN
	IF _stAxis.stStatus.bReadyToMove THEN
		fbMoveRelative.Execute := _stAxis.stStatus.bMoveRequested;
		IF _stAxis.stStatus.bMoveRequested THEN
			_stAxis.stStatus.bMoveRequested := FALSE;
		END_IF
	END_IF
END_IF

fbMoveRelative.Distance := _stAxis.stControl.fRelativePosition;
fbMoveRelative.Velocity := ABS(_stAxis.stControl.fVelocity);
fbMoveRelative.Acceleration := _stAxis.stControl.fAcceleration;
fbMoveRelative.Deceleration := _stAxis.stControl.fDeceleration;

fbMoveRelative(Axis := _stAxis.Axis);
fbMoveRelative.Execute := FALSE;

mMove_MoveRelative.Active := fbMoveRelative.Active;
mMove_MoveRelative.Done := fbMoveRelative.Done;
mMove_MoveRelative.Busy := fbMoveRelative.Busy;
mMove_MoveRelative.Error := fbMoveRelative.Error;
mMove_MoveRelative.ErrorID := fbMoveRelative.ErrorID;
mMove_MoveRelative.CommandAborted := fbMoveRelative.CommandAborted;

IF fbMoveRelative.Error THEN
    _stAxis.stError.nMoveRelativeErrorID := fbMoveRelative.ErrorID; //Set the error
END_IF
END_METHOD

METHOD mMove_MoveVelocity : ST_McStatus

IF _stAxis.stControl.eCommand = E_MotionFunctions.eMoveVelocity THEN
	IF _stAxis.stStatus.bReadyToMove THEN
		fbMoveVelocity.Execute := _stAxis.stStatus.bMoveRequested;
		IF _stAxis.stStatus.bMoveRequested THEN
			_stAxis.stStatus.bMoveRequested := FALSE;
		END_IF
	END_IF
END_IF

fbMoveVelocity.Direction := SEL(_stAxis.stControl.fVelocity < 0, MC_Positive_Direction, MC_Negative_Direction);
fbMoveVelocity.Velocity := ABS(_stAxis.stControl.fVelocity);

IF fbMoveVelocity.Execute THEN
	_stAxis.stControl.fVelocity := ABS(_stAxis.stControl.fVelocity);
END_IF

fbMoveVelocity.Acceleration := _stAxis.stControl.fAcceleration;
fbMoveVelocity.Deceleration := _stAxis.stControl.fDeceleration;

fbMoveVelocity(Axis := _stAxis.Axis);
fbMoveVelocity.Execute:= FALSE;

mMove_MoveVelocity.Active := fbMoveVelocity.Active;
mMove_MoveVelocity.InVelocity := fbMoveVelocity.InVelocity;
mMove_MoveVelocity.Busy := fbMoveVelocity.Busy;
mMove_MoveVelocity.Error := fbMoveVelocity.Error;
mMove_MoveVelocity.ErrorID := fbMoveVelocity.ErrorID;
mMove_MoveVelocity.CommandAborted := fbMoveVelocity.CommandAborted;

IF fbMoveVelocity.Error THEN
    _stAxis.stError.nMoveVelocityErrorID := fbMoveVelocity.ErrorID; //Set the error
END_IF
END_METHOD

METHOD mMove_SetPosition : ST_McStatus
IF _stAxis.stControl.eCommand = E_MotionFunctions.eSetPosition THEN
	fbSetPosition.Execute:= _stAxis.stControl.bExecute;
END_IF

fbSetPosition.Position:= _stAxis.stControl.fSetPosition;
fbSetPosition.Options.ClearPositionLag:= TRUE;

fbSetPosition(Axis := _stAxis.Axis);
fbSetPosition.Execute:= FALSE;

mMove_SetPosition.Busy := fbSetPosition.Busy;
mMove_SetPosition.Error := fbSetPosition.Error;
mMove_SetPosition.ErrorID := fbSetPosition.ErrorID;
mMove_SetPosition.Done := fbSetPosition.Done;

IF fbSetPosition.Error THEN
    _stAxis.stError.nSetPositionErrorID := fbSetPosition.ErrorID; //Set the error
END_IF
END_METHOD

METHOD mMove_Stop : ST_McStatus
fbStop.Deceleration := _stAxis.stControl.fDeceleration;
fbStop.Execute := _stAxis.stControl.bStop;

fbStop(Axis := _stAxis.Axis);

mMove_Stop.Busy := fbStop.Busy;
mMove_Stop.Done := fbStop.Done;
mMove_Stop.Error := fbStop.Error;
mMove_Stop.ErrorID := fbStop.ErrorID;
mMove_Stop.Active := fbStop.Active;
mMove_Stop.CommandAborted := fbStop.CommandAborted;

IF fbStop.Error THEN
    _stAxis.stError.nStopErrorID := fbStop.ErrorID; //Set the error
END_IF

//Execution of fbStop ended
fbStopFinishedRiseEdge(CLK:=fbStop.Done OR fbStop.Error OR fbStop.CommandAborted);
IF fbStopFinishedRiseEdge.Q THEN
    _stAxis.stControl.bStop := FALSE;
END_IF
END_METHOD

METHOD mParameters_Init : BOOL
IF _stAxis.stControl.bReinitialiseNcParameters THEN
	_stAxis.stStatus.bAxisInitialized := FALSE;
	_stAxis.stControl.bReinitialiseNcParameters := FALSE;
END_IF
IF _stAxis.stConfig.bReadMcParametersValid AND NOT _stAxis.stStatus.bAxisInitialized THEN
    _stAxis.stControl.fAcceleration := _stAxis.stConfig.fDefaultAcc;
    _stAxis.stControl.fDeceleration := _stAxis.stConfig.fDefaultDec;
    _stAxis.stControl.fVelocity := _stAxis.stConfig.fVelocityDefaultFast;
    _stAxis.stControl.fJogVelocity := _stAxis.stConfig.fVelocityDefaultSlow;

    _stAxis.stStatus.bAxisInitialized := TRUE;
END_IF
END_METHOD

METHOD mParameters_ReadNc : BOOL

(*This act reads the MC parameters using an MC_ReadParameter FB FOR each variable
Intended TO be executed once every PLC cycle
Another FB is used TO trasnfer default axis parameters TO the stAxisStruct so
bReadValid is used TO halt that trasnfer UNTIL the parameters have been
read successfully. It may take a couple OF cycles once the PLC starts up.*)


IF NOT _stAxis.stConfig.bReadMcParametersValid AND NOT fbReadAxisVeloManSlow.Valid THEN
	//Slow jogging Velocity
	fbReadAxisVeloManSlow(Axis := _stAxis.Axis,
                        Enable := TRUE,
                        ReadMode := READMODE_CYCLIC,
                        ParameterNumber := E_AxisParameters.AxisManualVelocitySlow,
                        Value => _stAxis.stConfig.fVelocityDefaultSlow);
END_IF

IF NOT _stAxis.stConfig.bReadMcParametersValid AND NOT fbReadAxisVeloManFast.Valid THEN
//Fast jogging velocity
fbReadAxisVeloManFast(Axis := _stAxis.Axis,
                        Enable := TRUE,
                        ReadMode := READMODE_CYCLIC,
                        ParameterNumber := E_AxisParameters.AxisManualVelocityFast,
                        Value => _stAxis.stConfig.fVelocityDefaultFast);
END_IF
IF NOT _stAxis.stConfig.bReadMcParametersValid AND NOT fbReadHomingVelToCam.Valid THEN
//Homing velocity to Cam
fbReadHomingVelToCam(Axis := _stAxis.Axis,
                        Enable := TRUE,
                        ReadMode := READMODE_CYCLIC,
                        ParameterNumber := E_AxisParameters.AxisVelocityToCam,
                        Value => _stAxis.stHomingConfig.fHomingVelToCam);
END_IF
IF NOT _stAxis.stConfig.bReadMcParametersValid AND NOT fbReadHomingVelFromCam.Valid THEN
//Homing velocity from Cam
fbReadHomingVelFromCam(Axis := _stAxis.Axis,
                        Enable := TRUE,
                        ReadMode := READMODE_CYCLIC,
                        ParameterNumber := E_AxisParameters.AxisVelocityFromCam,
                        Value => _stAxis.stHomingConfig.fHomingVelFromCam);
END_IF
IF NOT _stAxis.stConfig.bReadMcParametersValid AND NOT fbReadAxisVeloMax.Valid THEN
//Max velocity
fbReadAxisVeloMax(Axis := _stAxis.Axis,
                        Enable := TRUE,
                        ReadMode := READMODE_CYCLIC,
                        ParameterNumber := E_AxisParameters.AxisMaxVelocity,
                        Value => _stAxis.stConfig.fVeloMax);
END_IF
IF NOT _stAxis.stConfig.bReadMcParametersValid AND NOT fbReadAxisMaxAcc.Valid THEN
//Max acceleration
fbReadAxisMaxAcc(Axis := _stAxis.Axis,
                        Enable := TRUE,
                        ReadMode := READMODE_CYCLIC,
                        ParameterNumber := E_AxisParameters.AxisMaximumAcceleration,
                        Value => _stAxis.stConfig.fMaxAcc);
END_IF
IF NOT _stAxis.stConfig.bReadMcParametersValid AND NOT fbReadAxisMaxDec.Valid THEN
//Max deceleration
fbReadAxisMaxDec(Axis := _stAxis.Axis,
                        Enable := TRUE,
                        ReadMode := READMODE_CYCLIC,
                        ParameterNumber := E_AxisParameters.AxisMaximumDeceleration,
                        Value => _stAxis.stConfig.fMaxDec);
END_IF
IF NOT _stAxis.stConfig.bReadMcParametersValid AND NOT fbReadAxisAcc.Valid THEN
//Default acceleration
fbReadAxisAcc(Axis := _stAxis.Axis,
                        Enable := TRUE,
                        ReadMode := READMODE_CYCLIC,
                        ParameterNumber := E_AxisParameters.AxisDefaultAcceleration,
                        Value => _stAxis.stConfig.fDefaultAcc);
END_IF
IF NOT _stAxis.stConfig.bReadMcParametersValid AND NOT fbReadAxisDec.Valid THEN
//Default deceleration
fbReadAxisDec(Axis := _stAxis.Axis,
                        Enable := TRUE,
                        ReadMode := READMODE_CYCLIC,
                        ParameterNumber := E_AxisParameters.AxisDefaultDeceleration,
                        Value => _stAxis.stConfig.fDefaultDec);

END_IF
IF NOT _stAxis.stConfig.bReadMcParametersValid AND NOT fbReadEnMinSoftPosLimit.Valid THEN
//Soft limits enabled
fbReadEnMinSoftPosLimit(Axis := _stAxis.Axis,
                        Enable := TRUE,
                        ReadMode := READMODE_CYCLIC,
                        ParameterNumber := E_AxisParameters.EnableLimitBackward);
_stAxis.stConfig.bEnMinSoftPosLimit := LREAL_TO_BOOL(fbReadEnMinSoftPosLimit.Value);

END_IF
IF NOT _stAxis.stConfig.bReadMcParametersValid AND NOT fbReadEnMaxSoftPosLimit.Valid THEN
fbReadEnMaxSoftPosLimit(Axis := _stAxis.Axis,
                        Enable := TRUE,
                        ReadMode := READMODE_CYCLIC,
                        ParameterNumber := E_AxisParameters.EnableLimitForward);
_stAxis.stConfig.bEnMaxSoftPosLimit := LREAL_TO_BOOL(fbReadEnMaxSoftPosLimit.Value);

END_IF
IF NOT _stAxis.stConfig.bReadMcParametersValid AND NOT fbReadMinSoftPosLimit.Valid THEN
//Soft limit values
fbReadMinSoftPosLimit(Axis := _stAxis.Axis,
                        Enable := TRUE,
                        ReadMode := READMODE_CYCLIC,
                        ParameterNumber := E_AxisParameters.SWLimitBackward,
                        Value => _stAxis.stConfig.fMinSoftPosLimit);

END_IF
IF NOT _stAxis.stConfig.bReadMcParametersValid AND NOT fbReadMaxSoftPosLimit.Valid THEN
fbReadMaxSoftPosLimit(Axis := _stAxis.Axis,
                        Enable := TRUE,
                        ReadMode := READMODE_CYCLIC,
                        ParameterNumber := E_AxisParameters.SWLimitForward,
                        Value => _stAxis.stConfig.fMaxSoftPosLimit);

END_IF
IF NOT _stAxis.stConfig.bReadMcParametersValid AND NOT fbReadEnPositionLagMonitoring.Valid THEN
//Position Lag Monitoring
fbReadEnPositionLagMonitoring(Axis := _stAxis.Axis,
                        Enable := TRUE,
                        ReadMode := READMODE_CYCLIC,
                        ParameterNumber := E_AxisParameters.EnablePositionLagMonitoring);
_stAxis.stConfig.bEnPositionLagMonitoring := LREAL_TO_BOOL(fbReadEnPositionLagMonitoring.Value);

END_IF
IF NOT _stAxis.stConfig.bReadMcParametersValid AND NOT fbReadAxisMaxPosLagValue.Valid THEN
fbReadAxisMaxPosLagValue(Axis := _stAxis.Axis,
                        Enable := TRUE,
                        ReadMode := READMODE_CYCLIC,
                        ParameterNumber := E_AxisParameters.MaxPositionLag,
                        Value => _stAxis.stConfig.fMaxPosLagValue);

END_IF
IF NOT _stAxis.stConfig.bReadMcParametersValid AND NOT fbReadEnTargetPositionMonitoring.Valid THEN
// Target Position Monitoring
fbReadEnTargetPositionMonitoring(Axis := _stAxis.Axis,
                        Enable := TRUE,
                        ReadMode := READMODE_CYCLIC,
                        ParameterNumber := E_AxisParameters.SWLimitBackward);
_stAxis.stConfig.bEnTargetPositionMonitoring := LREAL_TO_BOOL(fbReadEnTargetPositionMonitoring.Value);

END_IF
IF NOT _stAxis.stConfig.bReadMcParametersValid AND NOT fbReadTargetPositionWindow.Valid THEN
fbReadTargetPositionWindow(Axis := _stAxis.Axis,
                        Enable := TRUE,
                        ReadMode := READMODE_CYCLIC,
                        ParameterNumber := E_AxisParameters.AxisTargetPositionWindow,
                        Value => _stAxis.stConfig.fTargetPositionWindow);
END_IF
//All variables are valid
_stAxis.stConfig.bReadMcParametersValid := FALSE;
_stAxis.stConfig.bReadMcParametersValid := fbReadAxisVeloManSlow.Valid AND
    fbReadAxisVeloManFast.Valid AND
    fbReadHomingVelToCam.Valid AND
    fbReadHomingVelFromCam.Valid AND
    fbReadAxisVeloMax.Valid AND
    fbReadAxisAcc.Valid AND
    fbReadAxisDec.Valid AND
    fbReadEnMinSoftPosLimit.Valid AND
    fbReadEnMaxSoftPosLimit.Valid AND
    fbReadMinSoftPosLimit.Valid AND
    fbReadMaxSoftPosLimit.Valid AND
    fbReadEnPositionLagMonitoring.Valid AND
    fbReadAxisMaxPosLagValue.Valid AND
    fbReadEnTargetPositionMonitoring.Valid AND
    fbReadTargetPositionWindow.Valid;

//One of the variables has a read error
_stAxis.stConfig.bReadMcParametersError := fbReadAxisVeloManSlow.Error OR
    fbReadAxisVeloManFast.Error OR
    fbReadHomingVelToCam.Error OR
    fbReadHomingVelFromCam.Error OR
    fbReadAxisVeloMax.Error OR
    fbReadAxisAcc.Error OR
    fbReadAxisDec.Error OR
    fbReadEnMinSoftPosLimit.Error OR
    fbReadEnMaxSoftPosLimit.Error OR
    fbReadMinSoftPosLimit.Error OR
    fbReadMaxSoftPosLimit.Error OR
    fbReadEnPositionLagMonitoring.Error OR
    fbReadAxisMaxPosLagValue.Error OR
    fbReadEnTargetPositionMonitoring.Error OR
    fbReadTargetPositionWindow.Error;
END_METHOD

METHOD mParameters_ReadParameter : ST_McStatus

IF _stAxis.stControl.eCommand = E_MotionFunctions.eReadParameter THEN
    fbReadParameter.Enable := _stAxis.stControl.bExecute;
END_IF

fbReadParameter.ReadMode := E_READMODE.READMODE_ONCE;
fbReadParameter.ParameterNumber := _stAxis.stConfig.eAxisParameters;

fbReadParameter(Axis := _stAxis.Axis);
fbReadParameter.Enable := FALSE;

